// TwinCAT 3 PLC project Lynus_Energy_MRTU
// Title: Lynus Energy ModbusRTU
// Company: Lynus AG
// ProjectVersion: 1.0.0.0
// ProgramVersion: 3.1.4024.12
// libraries:
//   Lynus Persistent Data V1, * (Lynus AG)
//   Lynus Standards, * (EfficientIO)
//   Tc2_Math, * (Beckhoff Automation GmbH)
//   Tc2_ModbusRTU, * (Beckhoff Automation GmbH)
//   Tc2_SerialCom, * (Beckhoff Automation GmbH)
//   Tc2_Standard, * (Beckhoff Automation GmbH)
//   Tc2_System, * (Beckhoff Automation GmbH)
//   Tc3_Module, * (Beckhoff Automation GmbH)
// project tree:
//   DUTs/Delta Inverter/ ST_DeltaPvInverter_Data.TcDUT
//   ENUMs/Delta Inverter/ eDeltaEvent.TcDUT, eDeltaOperatingState.TcDUT
//   ENUMs/Schrack/ E_Schrack_ECS_Error.TcDUT
//   FBs/Delta/ FB_Delta_PV_Inverter_Sunspec.TcPOU
//   FBs/Modbus RTU Master/ FB_KL6xxx_ModbusRTU_22B_Master.TcPOU
//   FBs/Schrack/ FB_ECS_Schrack_EM_CionHome.TcPOU

// ---- DUTs/Delta Inverter/ST_DeltaPvInverter_Data.TcDUT
TYPE ST_DeltaPvInverter_Data :
STRUCT
	eOperatingState			: eDeltaOperatingState;		//Operating State
	eEvent1					: eDeltaEvent;				//Eventfield
	rTotalMPPTPower			: REAL;						//Total DC Power in kW from the MPPT
	rCabinetTemp			: REAL;						//Cabinet Temperature
	rHeatSinkTemp			: REAL;						//Heat Sink Temperature
	arrCurrentFault			: ARRAY[1..8] OF WORD;		//Bit map for the current event of fault on inverter
	arrCurrentError			: ARRAY[1..5] OF WORD;		//Bit map for the current event of error on inverter
	arrCurrentWarning		: ARRAY[1..3] OF WORD;		//Bit map for the current event of warning on inverter
	arrMPPTPower			: ARRAY[1..6] OF REAL;		//Each MPPT DC Power in kW (Max 6 MPPT)
END_STRUCT
END_TYPE

// ---- ENUMs/Delta Inverter/eDeltaEvent.TcDUT
{attribute 'qualified_only'}
{attribute 'strict'}
TYPE eDeltaEvent :
(
	eNoInfo						:= 0,
	eGroundFault				:= 1,
	eDCOverVolt					:= 2,
	eACDisconnect				:= 3,
	eDCDisconnect				:= 4,
	eGridDisconnect				:= 5,
	eCabinetOpen				:= 6,
	eManualShutdown				:= 7,
	eOverTemp					:= 8,
	eOverFrequency				:= 9,
	eUnderFrequency				:= 10,
	eACOverVolt					:= 11,
	eACUnderVolt				:= 12,
	eBlownStringFuse			:= 13,
	eUnderTemp					:= 14,
	eMemoryLoss					:= 15,
	eHWTestFailure				:= 16,
	eOtherAlarm					:= 17,
	eOtherWarning				:= 18
);
END_TYPE

// ---- ENUMs/Delta Inverter/eDeltaOperatingState.TcDUT
{attribute 'qualified_only'}
{attribute 'strict'}
TYPE eDeltaOperatingState :
(
	eNoInfo				:= 0,
	eOff				:= 1,
	eSleeping			:= 2,
	eStarting			:= 3,
	eMppt				:= 4,
	eThrottled			:= 5,
	eShuttingDown		:= 6,
	eFault				:= 7,
	eStandby			:= 8
);
END_TYPE

// ---- ENUMs/Schrack/E_Schrack_ECS_Error.TcDUT
{attribute 'qualified_only'}
{attribute 'strict'}
TYPE E_Schrack_ECS_Error :
(
	eNoError := 0,
	eGroupError := 1,
	eFILSError := 2,
	eChargingCableError := 3,
	eChargingCableRejectedError := 4,
	eLoadContactorError := 5,
	eCommunicationErrorToTheCar := 6,
	eConfigurationErrorOnLP := 7,
	eRCMUError := 8,
	eRCMUErrorCurrentDetected := 9,
	eLockingError := 10,
	eUndervoltageError := 11,
	eOvervoltageError := 12,
	eControllerError := 13
);
END_TYPE

// ---- FBs/Delta/FB_Delta_PV_Inverter_Sunspec.TcPOU
FUNCTION_BLOCK FB_Delta_PV_Inverter_Sunspec
VAR_INPUT PERSISTENT
	bEnable										: BOOL;																			//{#lynus.ag#()} //Enable the Fuctionblock and his logic
	byMBAdress									: BYTE;																			//The Modbus Adress from the Slave
	diNrOfMBRTUMasterLine_IN					: DINT;																			//Number of the RTU Master Function on what this function can send or write data
END_VAR
VAR_OUTPUT
	stDeltaInverterData							: ST_DeltaPvInverter_Data;														//Structure with specific Delta Inverter Data
	stDataEMPower_PV							: ST_ElectricMeter_Output_Power;												//Output structure with Data from Electric Meter PV (Power Data)
	stDataEMCounter_PV							: ST_ElectricMeter_Output_Counter;												//Output structure with Data from Electric Meter PV (Counter Data)
	diNrOfEM_OUT_PV								: DINT;																			//Active Number from the Electric Meter for using on other functions
END_VAR
VAR
	{attribute 'hide'}
	fbElMeter									: FB_ElectricMeter;																//Electric Meter Function 
	{attribute 'hide'}
	fbNumberDevice								: FB_NumberOfDevice;															//Function block to calcualte the number of the Device
	{attribute 'hide'}
	timDelay									: TON;																			//Timer for Delay between Requests
	{attribute 'hide'}
	timTimeout									: TON;																			//Timer for Timeout
	{attribute 'hide'}
	timDissableFunctions						: TON;																			//Timer to dissable the Function after Lynus_Standards.Constants_General.tTimeDissableLynusFunctions Days without connection to the Lynus Cloud
	{attribute 'hide'}
	timResetConnectionOnGVL						: TON;																			//Timer to try reset the connection Flag on the GVL. (When somebody delete the Connection Function and make only a onlinechange)
	{attribute 'hide'}
	FPErrorMaster								: R_TRIG;																		//Internal positive Edge
	{attribute 'hide'}
	FPEnable									: R_TRIG;																		//Internal positive Edge
	{attribute 'hide'}
	fbConvertWord								: FB_CV_WORD_TO_DWORD;															//Convert 2 WORD in a DWORD
	{attribute 'hide'}
	arrPD										: ARRAY[1..5] OF FB_PersistentData_Number;										//Function to save persistent data
	{attribute 'hide'}
	arrDefaultModbusAdress						: ARRAY[1..247] OF BYTE;														//Default Modbuss Adress Array to fill in in the GVL Array after a Online change
	{attribute 'hide'}
	arrDefaultReadWrite							: ARRAY[1..Constants_Bussystems.wQuantityOfRegistersMBRTUMaster] OF WORD;		//Default Read/Write Array to fill in in the GVL Array after a Online change
	{attribute 'hide'}
	arrCounterForGVL							: ARRAY[1..2] OF DINT;															//Counter to clean old data on GVL
	{attribute 'hide'}
	bAdressIsSet								: BOOL;																			//Its true when the new Modbus Adress from the Slave is set in the Array on the GVL for the Master	
	{attribute 'hide'}
	bErrorInverter								: BOOL;																			//Error or Fault from Inverter
	{attribute 'hide'}
	bWarningInverter							: BOOL;																			//Warning from Inverter
	{attribute 'hide'}
	byWaitInStep								: BYTE;																			//Wait in Step before start to clean data on PLC
	{attribute 'hide'}
	byNumberOfSameMBAdress						: BYTE;																			//Number of Same Modbus adress on 1 Modbus Master
	{attribute 'hide'}
	byMBAdress_Old								: BYTE;																			//Old Modbus Adress to compare with the new Modbus Adress to start the state machine to set in the Array on the GVL
	{attribute 'hide'}
	byMBAdress_CP								: BYTE;																			//Variable to compare the Modbus Adress in the State Machine. When the Adress change when the state machine is active then the state machine starts from new with the new adress 
	{attribute 'hide'}
	byLPSlaveAdress								: BYTE;																			//Loop for the state machine to set the adress from the Slave in the array on the GVL
	{attribute 'hide'}
	byLPFillDefaultData							: BYTE;																			//Variable for Loop to fill default values in the Delta output structure
	{attribute 'hide'}
	byLPVendor64062								: BYTE;																			//Variable for Loop to fill the Error,Warning and Faults from Vendor 64062 to the Delta output structure
	{attribute 'hide'}
	iStateGVLData								: INT;																			//State machine to handle the data on the GVL
	{attribute 'hide'}
	iStateModbusRead							: INT;																			//State machine for read out Data over Modbus RTU
	{attribute 'hide'}
	iStateModbusError							: INT;																			//State machine for error out Data over Modbus RTU	
	{attribute 'hide'}
	iStateModbus_CP								: INT;																			//Variable to compare the state machine variable to set or reset the timeout timer
	{attribute 'hide'}
	iSFPowerMPPT								: INT;																			//Scale Factor for MPPT Power
	{attribute 'hide'}
	wNumberOfMPPT								: WORD;																			//Number of MPPT
	{attribute 'hide'}
	wLPCleanBuffer								: WORD;																			//Loop to clear the send and write Buffer on the GVL
	{attribute 'hide'}
	wLPPowerMPPT								: WORD;																			//Variable for Loop to fill the power for each MPPT in the output structure
	{attribute 'hide'}
	wNextModbusStartAdress						: WORD;																			//Next Modbus Start Adress why in Pic 160 the Number of Registers is variabel and so the next Modbus Registers in the next Pics can be different
	{attribute 'hide'}
	wNumberOfInputs								: WORD;																			//Number of Inputs from Pic 401 to calculate the Next Modbus Start Adress
	{attribute 'hide'}
	wPicID										: WORD;																			//ID of the PIC
	{attribute 'hide'}
	diNrOfMBRTUMasterLine_IN_Old				: DINT;																			//Old Modbus RTU Line to compare with the new Modbus RTU Line to start the state machine to set in the Array on the GVL
	{attribute 'hide'}
	diNrOfMBRTUMasterLine_IN_CP					: DINT;																			//Variable to compare the Modbus RTU Line in the State Machine. When the Modbus RTU Line change when the state machine is active then the state machine starts from new with the new Modbus RTU Line
	{attribute 'hide'}
	lrRestNextAdress							: LREAL;																		//Rest of the calculation for new Star Adress. In Sunspec each new PIC start with a even adress
END_VAR
VAR PERSISTENT
	{attribute 'conditionalshow'}
	byMBAdress_ForChange						: BYTE;																			//When we have 2 same Adresses on 1 Modbus RTU Line the byMBAdress_Int is set to 0. After a other change on the Input Adress Field so we can start to set the Adress in the Array in the GVL
	byMBAdress_Int								: BYTE;																			//Internal Adress what is using for the Read and Write functions
END_VAR

//Creator : Kai Ebensperger
//Company : Lynus AG
//Date : 26.10.2021
//Version : 1.0.0.0

//With this function its possible to read out values from the Delta PV Inverter over Modbus RTU
//The Protocoll is the Sunspec Protocol
//Versions that are supported : 1.16
//This Function use the INT+Scalfactor Format

//Infos for Operating State


//NOTE for diNr.....Designation => 
//_IN = Here Data come in from other Functions or go out to other functions about the GVL
//_OUT = Here Data go out to other functions about the GVL

(*--------------------------------------------------------------------------------------------Limits-------------------------------------------------------------------------------------*)

byMBAdress := LIMIT(0,byMBAdress,247);
	diNrOfMBRTUMasterLine_IN := LIMIT(0,diNrOfMBRTUMasterLine_IN,Constants_Bussystems.diMaxNumberOfMBRTUMasterKL6xxx);	

(*-------------------------------------------------------------Calcualte the number of ECS---------------------------------------------------------------*)

fbNumberDevice(
	diActualNumberOfDevices:= Lynus_Standards.GVL_Energy.stNumberOfDevices.diNumberOfElectricMeters, 
	diMaxNumberOfDevices:= Constants_Energy.diMaxNumberOfElectricMeters, 
	udiCounterOnlineChange:= TwinCAT_SystemInfoVarList._AppInfo.OnlineChangeCnt, 
	bNumberIsCalculatet=> , 
	bFPNumberIsCalculatet=> , 
	bOnlineChange=> , 
	diNumberForThisDevice=> diNrOfEM_OUT_PV, 
	diNumberOfTotalDevices=> );

//Write new Numer on GVL
IF fbNumberDevice.bFPNumberIsCalculatet THEN
	Lynus_Standards.GVL_Energy.stNumberOfDevices.diNumberOfElectricMeters := fbNumberDevice.diNumberOfTotalDevices;	
END_IF 

//Delete old Number on GVL
IF fbNumberDevice.bOnlineChange THEN 
	Lynus_Standards.GVL_Energy.stNumberOfDevices.diNumberOfElectricMeters := diNrOfEM_OUT_PV;	
		iStateGVLData := 1;	
			byMBAdress_Old := 0;
				diNrOfMBRTUMasterLine_IN_Old := 0;
END_IF

(*-------------------------------------------------------------Service from Backend is ready and check the connection to backen for dissabel/enable Function---------------------------------------------------------------*)

//Try to reset the variable for connection on the GVL. When all is normal then the Lynus Mqtt connection function set this variable to true in the next cycle
//When we have no connection to the backend then after Lynus_Standards.Constants_General.tTimeDissableLynusFunctions days the Function is dissabled with all of his functionalities
timResetConnectionOnGVL(IN:= NOT timResetConnectionOnGVL.Q, PT:= T#1H, Q=> , ET=> );
	IF timResetConnectionOnGVL.Q THEN Lynus_Standards.GVL_Communicator.bStateConnectionToEnableFunctions := FALSE; END_IF
		IF NOT Lynus_Standards.GVL_Communicator.bStateConnectionToEnableFunctions THEN timDissableFunctions.IN := TRUE; ELSE timDissableFunctions.IN := FALSE; END_IF  
			timDissableFunctions(IN:= , PT:= Lynus_Standards.Constants_General.tTimeDissableLynusFunctions, Q=> , ET=> );
			
(*--------------------------------------------------------------------------------------------Error from the Master Function-------------------------------------------------------------------------------------*)

FPErrorMaster(CLK:= Lynus_Standards.GVL_Bussystems.stDataOfMBRTUMasterKL6xxx[diNrOfMBRTUMasterLine_IN].byErrorWarning = 2 AND bEnable, Q=> );

(*--------------------------------------------------------------------------------------------Modbus Adress Slave Function-------------------------------------------------------------------------------------*)

FPEnable(CLK:= bEnable, Q=> );

//When the Adress is changed then set the new Adress in the Array
//When we have the Adress more then 1 time in 1 line then set to 0 and wait for the next change on the Input Variable for the Modbus Adress
IF byMBAdress <> byMBAdress_ForChange AND bEnable THEN byMBAdress_ForChange := byMBAdress; byNumberOfSameMBAdress := 0; END_IF     
	IF byMBAdress <> byMBAdress_Int AND byNumberOfSameMBAdress = 0 AND bEnable THEN byMBAdress_Int := byMBAdress; END_IF 
		IF NOT bEnable THEN byMBAdress_Int := 0; END_IF 
		
IF NOT Lynus_Standards.GVL_Bussystems.stDataOfMBRTUMasterKL6xxx[diNrOfMBRTUMasterLine_IN].bNoNewMBusAdress AND iStateGVLData = 0 AND (MEMCMP(ADR(byMBAdress_Int),ADR(byMBAdress_Old),SIZEOF(byMBAdress_Old)) <> 0 OR MEMCMP(ADR(diNrOfMBRTUMasterLine_IN),ADR(diNrOfMBRTUMasterLine_IN_Old),SIZEOF(diNrOfMBRTUMasterLine_IN_Old)) <> 0) THEN
	//Check if we have more then 1 time this Adress in 1 Line
	byNumberOfSameMBAdress := 0;	
		FOR byLPSlaveAdress := 1 TO 247 BY 1 DO
			IF Lynus_Standards.GVL_Bussystems.stDataOfMBRTUMasterKL6xxx[diNrOfMBRTUMasterLine_IN].arrAllModbusSlaveAdresses[byLPSlaveAdress] = byMBAdress_Int AND 
					Lynus_Standards.GVL_Bussystems.stDataOfMBRTUMasterKL6xxx[diNrOfMBRTUMasterLine_IN].arrAllModbusSlaveAdresses[byLPSlaveAdress] <> 0 THEN 
						byNumberOfSameMBAdress := byNumberOfSameMBAdress + 1; 
				END_IF 
		END_FOR
			IF byNumberOfSameMBAdress > 0 THEN 
				byMBAdress_Int := 0;
			END_IF	
				bAdressIsSet := FALSE; 
					//Delte the old Adress from the old Array
					FOR byLPSlaveAdress := 1 TO 247 BY 1 DO
						IF Lynus_Standards.GVL_Bussystems.stDataOfMBRTUMasterKL6xxx[diNrOfMBRTUMasterLine_IN_Old].arrAllModbusSlaveAdresses[byLPSlaveAdress] = byMBAdress_Old THEN
							Lynus_Standards.GVL_Bussystems.stDataOfMBRTUMasterKL6xxx[diNrOfMBRTUMasterLine_IN_Old].arrAllModbusSlaveAdresses[byLPSlaveAdress] := 0;
						END_IF	 
					END_FOR
						//Set the New Adress in Array
						byMBAdress_Old := byMBAdress_Int;
							diNrOfMBRTUMasterLine_IN_Old := diNrOfMBRTUMasterLine_IN;
								FOR byLPSlaveAdress := 1 TO 247 BY 1 DO
									IF Lynus_Standards.GVL_Bussystems.stDataOfMBRTUMasterKL6xxx[diNrOfMBRTUMasterLine_IN].arrAllModbusSlaveAdresses[byLPSlaveAdress] = 0 AND NOT bAdressIsSet THEN 
										Lynus_Standards.GVL_Bussystems.stDataOfMBRTUMasterKL6xxx[diNrOfMBRTUMasterLine_IN].arrAllModbusSlaveAdresses[byLPSlaveAdress] := byMBAdress_Int; 
											bAdressIsSet := TRUE;
									END_IF 
								END_FOR
END_IF	

(*--------------------------------------------------------------------------------------------State Machine Read--------------------------------------------------------------------------------------*)

//Timer for Delay
timDelay(IN:= , PT:= T#250MS, Q=> , ET=> );

//Timer for Timeout in Statemachine
IF iStateModbusRead > 0 AND iStateModbusRead <= 8 AND iStateModbusRead = iStateModbus_CP THEN
		timTimeout.IN := TRUE;
ELSE	
		timTimeout.IN := FALSE;
END_IF
	//Timeout Timer is dissabled when the slave wait that his adress is in porgress on the RTU Master, or is dissabled or the Terminal is not configured
	IF iStateModbusRead = 0 OR NOT bEnable OR NOT Lynus_Standards.GVL_Bussystems.stDataOfMBRTUMasterKL6xxx[diNrOfMBRTUMasterLine_IN].bTerminalIsConfigured THEN timTimeout.IN := FALSE; END_IF
		timTimeout(IN:= , PT:= T#15S, Q=> , ET=> );

//Not Enabled
IF NOT bEnable OR NOT Lynus_Standards.GVL_Bussystems.stDataOfMBRTUMasterKL6xxx[diNrOfMBRTUMasterLine_IN].bTerminalIsConfigured THEN iStateModbusRead := 0; iStateModbusError := 0; END_IF		
		
CASE iStateModbusRead OF

	0://Init Step (Wait that the Slave is enabled and the Terminal is configured)
		
		//Set Delta Output Structure to default
		IF NOT bEnable OR NOT Lynus_Standards.GVL_Bussystems.stDataOfMBRTUMasterKL6xxx[diNrOfMBRTUMasterLine_IN].bTerminalIsConfigured THEN 
			stDeltaInverterData.rTotalMPPTPower := 0;
				stDeltaInverterData.rCabinetTemp := 0;
					stDeltaInverterData.rHeatSinkTemp := 0;
						FOR byLPFillDefaultData := 1 TO 6 BY 1 DO
							stDeltaInverterData.arrMPPTPower[byLPFillDefaultData] := 0;
						END_FOR
							stDeltaInverterData.eEvent1 := eDeltaEvent.eNoInfo;
								stDeltaInverterData.eOperatingState := eDeltaOperatingState.eNoInfo;
		END_IF
		
		iSFPowerMPPT := 0;
			wNumberOfMPPT := 0;
				wNextModbusStartAdress := 0;
					wNumberOfInputs := 0;
						lrRestNextAdress := 0;
				
		IF bEnable AND Lynus_Standards.GVL_Bussystems.stDataOfMBRTUMasterKL6xxx[diNrOfMBRTUMasterLine_IN].bTerminalIsConfigured THEN
			//Start Timer for start the Statemachine
			IF NOT Lynus_Standards.GVL_Bussystems.stDataOfMBRTUMasterKL6xxx[diNrOfMBRTUMasterLine_IN].bMasterIsBusy THEN timDelay.IN := TRUE; END_IF 
		
			//Reset the Read and Write Buffer on the GVL before starting
			IF byMBAdress_Int = Lynus_Standards.GVL_Bussystems.stDataOfMBRTUMasterKL6xxx[diNrOfMBRTUMasterLine_IN].byActualMBAdressInProgrss THEN
				FOR wLPCleanBuffer := 1 TO Constants_Bussystems.wQuantityOfRegistersMBRTUMaster BY 1 DO
					Lynus_Standards.GVL_Bussystems.stDataOfMBRTUMasterKL6xxx[diNrOfMBRTUMasterLine_IN].arrReadOutData[wLPCleanBuffer] := 0;
						Lynus_Standards.GVL_Bussystems.stDataOfMBRTUMasterKL6xxx[diNrOfMBRTUMasterLine_IN].arrWriteOutData[wLPCleanBuffer] := 0;
				END_FOR
			END_IF
			
			IF timDelay.Q AND byMBAdress_Int = Lynus_Standards.GVL_Bussystems.stDataOfMBRTUMasterKL6xxx[diNrOfMBRTUMasterLine_IN].byActualMBAdressInProgrss AND NOT Lynus_Standards.GVL_Bussystems.stDataOfMBRTUMasterKL6xxx[diNrOfMBRTUMasterLine_IN].bReadWriteIsDone THEN
				timDelay.IN := FALSE;
					iStateModbusRead := 1;
						diNrOfMBRTUMasterLine_IN_CP := diNrOfMBRTUMasterLine_IN;
							byMBAdress_CP := byMBAdress_Int; 	
								Lynus_Standards.GVL_Bussystems.stDataOfMBRTUMasterKL6xxx[diNrOfMBRTUMasterLine_IN].bSlaveStartReadOrWrite := FALSE;
			END_IF
		END_IF
	
	1://Read Out Values from Pic 103 of the Sunspec Protocol (Register 40084)
		iStateModbus_CP := iStateModbusRead;
		
		Lynus_Standards.GVL_Bussystems.stDataOfMBRTUMasterKL6xxx[diNrOfMBRTUMasterLine_IN].eMBRTUReadWriteMode := E_MBRTUMaster_ReadWriteMode.eModbusRTUMaster_ReadRegs;
			Lynus_Standards.GVL_Bussystems.stDataOfMBRTUMasterKL6xxx[diNrOfMBRTUMasterLine_IN].wNumberOfRegister := 39;
				Lynus_Standards.GVL_Bussystems.stDataOfMBRTUMasterKL6xxx[diNrOfMBRTUMasterLine_IN].wModbusRegister := 40073;
		
		IF NOT Lynus_Standards.GVL_Bussystems.stDataOfMBRTUMasterKL6xxx[diNrOfMBRTUMasterLine_IN].bMasterIsBusy THEN timDelay.IN := TRUE; END_IF 

		//Copy the read out Data
		IF NOT Lynus_Standards.GVL_Bussystems.stDataOfMBRTUMasterKL6xxx[diNrOfMBRTUMasterLine_IN].bMasterIsBusy AND Lynus_Standards.GVL_Bussystems.stDataOfMBRTUMasterKL6xxx[diNrOfMBRTUMasterLine_IN].byErrorWarning = 0 AND timDelay.Q AND diNrOfMBRTUMasterLine_IN = diNrOfMBRTUMasterLine_IN_CP AND byMBAdress_Int = byMBAdress_CP THEN
			//Current L1
			IF WORD_TO_INT(Lynus_Standards.GVL_Bussystems.stDataOfMBRTUMasterKL6xxx[diNrOfMBRTUMasterLine_IN].arrReadOutData[4]) >= - 10 AND WORD_TO_INT(Lynus_Standards.GVL_Bussystems.stDataOfMBRTUMasterKL6xxx[diNrOfMBRTUMasterLine_IN].arrReadOutData[4]) <= 10 THEN
				fbElMeter.lrCurrentL1 := Lynus_Standards.GVL_Bussystems.stDataOfMBRTUMasterKL6xxx[diNrOfMBRTUMasterLine_IN].arrReadOutData[1] * EXPT(10,WORD_TO_INT(Lynus_Standards.GVL_Bussystems.stDataOfMBRTUMasterKL6xxx[diNrOfMBRTUMasterLine_IN].arrReadOutData[4]));
			END_IF
			//Current L2
			IF WORD_TO_INT(Lynus_Standards.GVL_Bussystems.stDataOfMBRTUMasterKL6xxx[diNrOfMBRTUMasterLine_IN].arrReadOutData[4]) >= - 10 AND WORD_TO_INT(Lynus_Standards.GVL_Bussystems.stDataOfMBRTUMasterKL6xxx[diNrOfMBRTUMasterLine_IN].arrReadOutData[4]) <= 10 THEN
				fbElMeter.lrCurrentL2 := Lynus_Standards.GVL_Bussystems.stDataOfMBRTUMasterKL6xxx[diNrOfMBRTUMasterLine_IN].arrReadOutData[2] * EXPT(10,WORD_TO_INT(Lynus_Standards.GVL_Bussystems.stDataOfMBRTUMasterKL6xxx[diNrOfMBRTUMasterLine_IN].arrReadOutData[4]));
			END_IF
			//Current L3
			IF WORD_TO_INT(Lynus_Standards.GVL_Bussystems.stDataOfMBRTUMasterKL6xxx[diNrOfMBRTUMasterLine_IN].arrReadOutData[4]) >= - 10 AND WORD_TO_INT(Lynus_Standards.GVL_Bussystems.stDataOfMBRTUMasterKL6xxx[diNrOfMBRTUMasterLine_IN].arrReadOutData[4]) <= 10 THEN
				fbElMeter.lrCurrentL3 := Lynus_Standards.GVL_Bussystems.stDataOfMBRTUMasterKL6xxx[diNrOfMBRTUMasterLine_IN].arrReadOutData[3] * EXPT(10,WORD_TO_INT(Lynus_Standards.GVL_Bussystems.stDataOfMBRTUMasterKL6xxx[diNrOfMBRTUMasterLine_IN].arrReadOutData[4]));
			END_IF
			//Voltage L1/N
			IF WORD_TO_INT(Lynus_Standards.GVL_Bussystems.stDataOfMBRTUMasterKL6xxx[diNrOfMBRTUMasterLine_IN].arrReadOutData[11]) >= - 10 AND WORD_TO_INT(Lynus_Standards.GVL_Bussystems.stDataOfMBRTUMasterKL6xxx[diNrOfMBRTUMasterLine_IN].arrReadOutData[11]) <= 10 THEN
				fbElMeter.lrVoltageL1N := Lynus_Standards.GVL_Bussystems.stDataOfMBRTUMasterKL6xxx[diNrOfMBRTUMasterLine_IN].arrReadOutData[8] * EXPT(10,WORD_TO_INT(Lynus_Standards.GVL_Bussystems.stDataOfMBRTUMasterKL6xxx[diNrOfMBRTUMasterLine_IN].arrReadOutData[11]));
			END_IF
			//Voltage L2/N
			IF WORD_TO_INT(Lynus_Standards.GVL_Bussystems.stDataOfMBRTUMasterKL6xxx[diNrOfMBRTUMasterLine_IN].arrReadOutData[11]) >= - 10 AND WORD_TO_INT(Lynus_Standards.GVL_Bussystems.stDataOfMBRTUMasterKL6xxx[diNrOfMBRTUMasterLine_IN].arrReadOutData[11]) <= 10 THEN
				fbElMeter.lrVoltageL2N := Lynus_Standards.GVL_Bussystems.stDataOfMBRTUMasterKL6xxx[diNrOfMBRTUMasterLine_IN].arrReadOutData[9] * EXPT(10,WORD_TO_INT(Lynus_Standards.GVL_Bussystems.stDataOfMBRTUMasterKL6xxx[diNrOfMBRTUMasterLine_IN].arrReadOutData[11]));
			END_IF
			//Voltage L3/N
			IF WORD_TO_INT(Lynus_Standards.GVL_Bussystems.stDataOfMBRTUMasterKL6xxx[diNrOfMBRTUMasterLine_IN].arrReadOutData[11]) >= - 10 AND WORD_TO_INT(Lynus_Standards.GVL_Bussystems.stDataOfMBRTUMasterKL6xxx[diNrOfMBRTUMasterLine_IN].arrReadOutData[11]) <= 10 THEN
				fbElMeter.lrVoltageL3N := Lynus_Standards.GVL_Bussystems.stDataOfMBRTUMasterKL6xxx[diNrOfMBRTUMasterLine_IN].arrReadOutData[10] * EXPT(10,WORD_TO_INT(Lynus_Standards.GVL_Bussystems.stDataOfMBRTUMasterKL6xxx[diNrOfMBRTUMasterLine_IN].arrReadOutData[11]));
			END_IF
			//AC Power
			IF WORD_TO_INT(Lynus_Standards.GVL_Bussystems.stDataOfMBRTUMasterKL6xxx[diNrOfMBRTUMasterLine_IN].arrReadOutData[13]) >= - 10 AND WORD_TO_INT(Lynus_Standards.GVL_Bussystems.stDataOfMBRTUMasterKL6xxx[diNrOfMBRTUMasterLine_IN].arrReadOutData[13]) <= 10 THEN  
				fbElMeter.lrPowerTotal := WORD_TO_INT(Lynus_Standards.GVL_Bussystems.stDataOfMBRTUMasterKL6xxx[diNrOfMBRTUMasterLine_IN].arrReadOutData[12]) * EXPT(10,WORD_TO_INT(Lynus_Standards.GVL_Bussystems.stDataOfMBRTUMasterKL6xxx[diNrOfMBRTUMasterLine_IN].arrReadOutData[13]));
			END_IF
			//Hz
			IF WORD_TO_INT(Lynus_Standards.GVL_Bussystems.stDataOfMBRTUMasterKL6xxx[diNrOfMBRTUMasterLine_IN].arrReadOutData[15]) >= - 10 AND WORD_TO_INT(Lynus_Standards.GVL_Bussystems.stDataOfMBRTUMasterKL6xxx[diNrOfMBRTUMasterLine_IN].arrReadOutData[15]) <= 10 THEN  
				fbElMeter.lrFrequency := Lynus_Standards.GVL_Bussystems.stDataOfMBRTUMasterKL6xxx[diNrOfMBRTUMasterLine_IN].arrReadOutData[14] * EXPT(10,WORD_TO_INT(Lynus_Standards.GVL_Bussystems.stDataOfMBRTUMasterKL6xxx[diNrOfMBRTUMasterLine_IN].arrReadOutData[15]));
			END_IF
			//Apparent Power
			IF WORD_TO_INT(Lynus_Standards.GVL_Bussystems.stDataOfMBRTUMasterKL6xxx[diNrOfMBRTUMasterLine_IN].arrReadOutData[17]) >= - 10 AND WORD_TO_INT(Lynus_Standards.GVL_Bussystems.stDataOfMBRTUMasterKL6xxx[diNrOfMBRTUMasterLine_IN].arrReadOutData[17]) <= 10 THEN  
				fbElMeter.lrApparentPowerTotal := WORD_TO_INT(Lynus_Standards.GVL_Bussystems.stDataOfMBRTUMasterKL6xxx[diNrOfMBRTUMasterLine_IN].arrReadOutData[16]) * EXPT(10,WORD_TO_INT(Lynus_Standards.GVL_Bussystems.stDataOfMBRTUMasterKL6xxx[diNrOfMBRTUMasterLine_IN].arrReadOutData[17]));
			END_IF
			//Reactive Power
			IF WORD_TO_INT(Lynus_Standards.GVL_Bussystems.stDataOfMBRTUMasterKL6xxx[diNrOfMBRTUMasterLine_IN].arrReadOutData[19]) >= - 10 AND WORD_TO_INT(Lynus_Standards.GVL_Bussystems.stDataOfMBRTUMasterKL6xxx[diNrOfMBRTUMasterLine_IN].arrReadOutData[19]) <= 10 THEN  
				fbElMeter.lrReactivePowerTotal := WORD_TO_INT(Lynus_Standards.GVL_Bussystems.stDataOfMBRTUMasterKL6xxx[diNrOfMBRTUMasterLine_IN].arrReadOutData[18]) * EXPT(10,WORD_TO_INT(Lynus_Standards.GVL_Bussystems.stDataOfMBRTUMasterKL6xxx[diNrOfMBRTUMasterLine_IN].arrReadOutData[19]));
			END_IF
			//Produced Energy
			IF WORD_TO_INT(Lynus_Standards.GVL_Bussystems.stDataOfMBRTUMasterKL6xxx[diNrOfMBRTUMasterLine_IN].arrReadOutData[24]) >= - 10 AND WORD_TO_INT(Lynus_Standards.GVL_Bussystems.stDataOfMBRTUMasterKL6xxx[diNrOfMBRTUMasterLine_IN].arrReadOutData[24]) <= 10 THEN  
				fbConvertWord(wInputValue_1:= Lynus_Standards.GVL_Bussystems.stDataOfMBRTUMasterKL6xxx[diNrOfMBRTUMasterLine_IN].arrReadOutData[22], wInputValue_2:= Lynus_Standards.GVL_Bussystems.stDataOfMBRTUMasterKL6xxx[diNrOfMBRTUMasterLine_IN].arrReadOutData[23], eByteOrderForConvert:= eByteOrder.eBigEndian, dwOutputValue=> );
					fbElMeter.lrCounterEnergyT1_Production := fbConvertWord.dwOutputValue * EXPT(10,WORD_TO_INT(Lynus_Standards.GVL_Bussystems.stDataOfMBRTUMasterKL6xxx[diNrOfMBRTUMasterLine_IN].arrReadOutData[24]));
						fbElMeter.lrCounterEnergyT1_Production := fbElMeter.lrCounterEnergyT1_Production / 1000;
							fbElMeter.lrTotalCounterEnergy_Production := fbElMeter.lrCounterEnergyT1_Production; 	
			END_IF
			//Cabinet Temperature
			IF WORD_TO_INT(Lynus_Standards.GVL_Bussystems.stDataOfMBRTUMasterKL6xxx[diNrOfMBRTUMasterLine_IN].arrReadOutData[35]) >= - 10 AND WORD_TO_INT(Lynus_Standards.GVL_Bussystems.stDataOfMBRTUMasterKL6xxx[diNrOfMBRTUMasterLine_IN].arrReadOutData[35]) <= 10 THEN  
				stDeltaInverterData.rCabinetTemp := LREAL_TO_REAL(WORD_TO_INT(Lynus_Standards.GVL_Bussystems.stDataOfMBRTUMasterKL6xxx[diNrOfMBRTUMasterLine_IN].arrReadOutData[31]) * EXPT(10,WORD_TO_INT(Lynus_Standards.GVL_Bussystems.stDataOfMBRTUMasterKL6xxx[diNrOfMBRTUMasterLine_IN].arrReadOutData[35])));
			END_IF
			//Heat Sink Temperature
			IF WORD_TO_INT(Lynus_Standards.GVL_Bussystems.stDataOfMBRTUMasterKL6xxx[diNrOfMBRTUMasterLine_IN].arrReadOutData[35]) >= - 10 AND WORD_TO_INT(Lynus_Standards.GVL_Bussystems.stDataOfMBRTUMasterKL6xxx[diNrOfMBRTUMasterLine_IN].arrReadOutData[35]) <= 10 THEN  
				stDeltaInverterData.rHeatSinkTemp := LREAL_TO_REAL(WORD_TO_INT(Lynus_Standards.GVL_Bussystems.stDataOfMBRTUMasterKL6xxx[diNrOfMBRTUMasterLine_IN].arrReadOutData[32]) * EXPT(10,WORD_TO_INT(Lynus_Standards.GVL_Bussystems.stDataOfMBRTUMasterKL6xxx[diNrOfMBRTUMasterLine_IN].arrReadOutData[35])));
			END_IF
			//Operating State
			stDeltaInverterData.eOperatingState := eDeltaOperatingState.eNoInfo;
			IF Lynus_Standards.GVL_Bussystems.stDataOfMBRTUMasterKL6xxx[diNrOfMBRTUMasterLine_IN].arrReadOutData[36] = 1 THEN stDeltaInverterData.eOperatingState := eDeltaOperatingState.eOff;
			ELSIF Lynus_Standards.GVL_Bussystems.stDataOfMBRTUMasterKL6xxx[diNrOfMBRTUMasterLine_IN].arrReadOutData[36] = 2 THEN stDeltaInverterData.eOperatingState := eDeltaOperatingState.eSleeping;
			ELSIF Lynus_Standards.GVL_Bussystems.stDataOfMBRTUMasterKL6xxx[diNrOfMBRTUMasterLine_IN].arrReadOutData[36] = 3 THEN stDeltaInverterData.eOperatingState := eDeltaOperatingState.eStarting;
			ELSIF Lynus_Standards.GVL_Bussystems.stDataOfMBRTUMasterKL6xxx[diNrOfMBRTUMasterLine_IN].arrReadOutData[36] = 4 THEN stDeltaInverterData.eOperatingState := eDeltaOperatingState.eMppt;
			ELSIF Lynus_Standards.GVL_Bussystems.stDataOfMBRTUMasterKL6xxx[diNrOfMBRTUMasterLine_IN].arrReadOutData[36] = 5 THEN stDeltaInverterData.eOperatingState := eDeltaOperatingState.eThrottled;
			ELSIF Lynus_Standards.GVL_Bussystems.stDataOfMBRTUMasterKL6xxx[diNrOfMBRTUMasterLine_IN].arrReadOutData[36] = 6 THEN stDeltaInverterData.eOperatingState := eDeltaOperatingState.eShuttingDown;
			ELSIF Lynus_Standards.GVL_Bussystems.stDataOfMBRTUMasterKL6xxx[diNrOfMBRTUMasterLine_IN].arrReadOutData[36] = 7 THEN stDeltaInverterData.eOperatingState := eDeltaOperatingState.eFault;
			ELSIF Lynus_Standards.GVL_Bussystems.stDataOfMBRTUMasterKL6xxx[diNrOfMBRTUMasterLine_IN].arrReadOutData[36] = 8 THEN stDeltaInverterData.eOperatingState := eDeltaOperatingState.eStandby;
			END_IF 
			//Event 1
			fbConvertWord(wInputValue_1:= Lynus_Standards.GVL_Bussystems.stDataOfMBRTUMasterKL6xxx[diNrOfMBRTUMasterLine_IN].arrReadOutData[38], wInputValue_2:= Lynus_Standards.GVL_Bussystems.stDataOfMBRTUMasterKL6xxx[diNrOfMBRTUMasterLine_IN].arrReadOutData[39], eByteOrderForConvert:= eByteOrder.eBigEndian, dwOutputValue=> );
			stDeltaInverterData.eEvent1 := eDeltaEvent.eNoInfo;
			IF fbConvertWord.dwOutputValue.0 THEN stDeltaInverterData.eEvent1 := eDeltaEvent.eGroundFault;
			ELSIF fbConvertWord.dwOutputValue.1 THEN stDeltaInverterData.eEvent1 := eDeltaEvent.eDCOverVolt;
			ELSIF fbConvertWord.dwOutputValue.2 THEN stDeltaInverterData.eEvent1 := eDeltaEvent.eACDisconnect;
			ELSIF fbConvertWord.dwOutputValue.3 THEN stDeltaInverterData.eEvent1 := eDeltaEvent.eDCDisconnect;
			ELSIF fbConvertWord.dwOutputValue.4 THEN stDeltaInverterData.eEvent1 := eDeltaEvent.eGridDisconnect;
			ELSIF fbConvertWord.dwOutputValue.5 THEN stDeltaInverterData.eEvent1 := eDeltaEvent.eCabinetOpen;
			ELSIF fbConvertWord.dwOutputValue.6 THEN stDeltaInverterData.eEvent1 := eDeltaEvent.eManualShutdown;
			ELSIF fbConvertWord.dwOutputValue.7 THEN stDeltaInverterData.eEvent1 := eDeltaEvent.eOverTemp;
			ELSIF fbConvertWord.dwOutputValue.8 THEN stDeltaInverterData.eEvent1 := eDeltaEvent.eOverFrequency;
			ELSIF fbConvertWord.dwOutputValue.9 THEN stDeltaInverterData.eEvent1 := eDeltaEvent.eUnderFrequency;
			ELSIF fbConvertWord.dwOutputValue.10 THEN stDeltaInverterData.eEvent1 := eDeltaEvent.eACOverVolt;
			ELSIF fbConvertWord.dwOutputValue.11 THEN stDeltaInverterData.eEvent1 := eDeltaEvent.eACUnderVolt;
			ELSIF fbConvertWord.dwOutputValue.12 THEN stDeltaInverterData.eEvent1 := eDeltaEvent.eBlownStringFuse;
			ELSIF fbConvertWord.dwOutputValue.13 THEN stDeltaInverterData.eEvent1 := eDeltaEvent.eUnderTemp;
			ELSIF fbConvertWord.dwOutputValue.14 THEN stDeltaInverterData.eEvent1 := eDeltaEvent.eMemoryLoss;
			ELSIF fbConvertWord.dwOutputValue.15 THEN stDeltaInverterData.eEvent1 := eDeltaEvent.eHWTestFailure;
			ELSIF fbConvertWord.dwOutputValue.16 THEN stDeltaInverterData.eEvent1 := eDeltaEvent.eOtherAlarm;
			ELSIF fbConvertWord.dwOutputValue.17 THEN stDeltaInverterData.eEvent1 := eDeltaEvent.eOtherWarning;	
			END_IF
		END_IF     				
		
		//Send the Read or Write Command to the Master
		Lynus_Standards.GVL_Bussystems.stDataOfMBRTUMasterKL6xxx[diNrOfMBRTUMasterLine_IN].bSlaveStartReadOrWrite := TRUE;
		
		//Go to the Next Step
		IF NOT Lynus_Standards.GVL_Bussystems.stDataOfMBRTUMasterKL6xxx[diNrOfMBRTUMasterLine_IN].bMasterIsBusy AND Lynus_Standards.GVL_Bussystems.stDataOfMBRTUMasterKL6xxx[diNrOfMBRTUMasterLine_IN].byErrorWarning = 0 AND timDelay.Q AND 
			diNrOfMBRTUMasterLine_IN = diNrOfMBRTUMasterLine_IN_CP AND byMBAdress_Int = byMBAdress_CP AND NOT timTimeout.Q THEN
				timDelay.IN := FALSE;
					Lynus_Standards.GVL_Bussystems.stDataOfMBRTUMasterKL6xxx[diNrOfMBRTUMasterLine_IN].bSlaveStartReadOrWrite := FALSE;
						iStateModbusRead := 2;
							wNextModbusStartAdress := 40122;		
		END_IF

			//Error on Master, changes on Inputs or Timeout
		 	IF timTimeout.Q OR diNrOfMBRTUMasterLine_IN <> diNrOfMBRTUMasterLine_IN_CP OR byMBAdress_Int <> byMBAdress_CP OR FPErrorMaster.Q THEN 
				iStateModbusError := 300; 
					diNrOfMBRTUMasterLine_IN_CP := diNrOfMBRTUMasterLine_IN; 
						byMBAdress_CP := byMBAdress_Int; 
			END_IF 
	
	2://Read Out Values from Pic 120 to Start Adress for PIC 160 of the Sunspec Protocoll		
		iStateModbus_CP := iStateModbusRead;
		
		Lynus_Standards.GVL_Bussystems.stDataOfMBRTUMasterKL6xxx[diNrOfMBRTUMasterLine_IN].eMBRTUReadWriteMode := E_MBRTUMaster_ReadWriteMode.eModbusRTUMaster_ReadRegs;
			Lynus_Standards.GVL_Bussystems.stDataOfMBRTUMasterKL6xxx[diNrOfMBRTUMasterLine_IN].wNumberOfRegister := 2;
				Lynus_Standards.GVL_Bussystems.stDataOfMBRTUMasterKL6xxx[diNrOfMBRTUMasterLine_IN].wModbusRegister := wNextModbusStartAdress;
		
		IF NOT Lynus_Standards.GVL_Bussystems.stDataOfMBRTUMasterKL6xxx[diNrOfMBRTUMasterLine_IN].bMasterIsBusy THEN timDelay.IN := TRUE; END_IF 

		//Copy the read out Data
		IF NOT Lynus_Standards.GVL_Bussystems.stDataOfMBRTUMasterKL6xxx[diNrOfMBRTUMasterLine_IN].bMasterIsBusy AND Lynus_Standards.GVL_Bussystems.stDataOfMBRTUMasterKL6xxx[diNrOfMBRTUMasterLine_IN].byErrorWarning = 0 AND timDelay.Q AND diNrOfMBRTUMasterLine_IN = diNrOfMBRTUMasterLine_IN_CP AND byMBAdress_Int = byMBAdress_CP THEN
			//PIC ID
			wPicID := Lynus_Standards.GVL_Bussystems.stDataOfMBRTUMasterKL6xxx[diNrOfMBRTUMasterLine_IN].arrReadOutData[1];
			//Number of Inputs
			wNumberOfInputs := Lynus_Standards.GVL_Bussystems.stDataOfMBRTUMasterKL6xxx[diNrOfMBRTUMasterLine_IN].arrReadOutData[2];
		END_IF     					
		
		//Send the Read or Write Command to the Master
		Lynus_Standards.GVL_Bussystems.stDataOfMBRTUMasterKL6xxx[diNrOfMBRTUMasterLine_IN].bSlaveStartReadOrWrite := TRUE;
		
		//Go to the Next Step
		IF NOT Lynus_Standards.GVL_Bussystems.stDataOfMBRTUMasterKL6xxx[diNrOfMBRTUMasterLine_IN].bMasterIsBusy AND Lynus_Standards.GVL_Bussystems.stDataOfMBRTUMasterKL6xxx[diNrOfMBRTUMasterLine_IN].byErrorWarning = 0 AND timDelay.Q AND 
			diNrOfMBRTUMasterLine_IN = diNrOfMBRTUMasterLine_IN_CP AND byMBAdress_Int = byMBAdress_CP AND NOT timTimeout.Q THEN
				timDelay.IN := FALSE;
					Lynus_Standards.GVL_Bussystems.stDataOfMBRTUMasterKL6xxx[diNrOfMBRTUMasterLine_IN].bSlaveStartReadOrWrite := FALSE;
						iStateModbusRead := 3;	
							lrRestNextAdress := 0;
			//Calculate next Modbus Start Adress for next Pic
			wNextModbusStartAdress := wNextModbusStartAdress + wNumberOfInputs + 2;
				lrRestNextAdress := FRAC(WORD_TO_REAL(wNextModbusStartAdress) / 2);	
					//If it ends with an odd number, the next PIC starts with an even address
					IF lrRestNextAdress <> 0 THEN wNextModbusStartAdress := wNextModbusStartAdress + 1; END_IF 
		END_IF

			//Error on Master, changes on Inputs or Timeout
		 	IF timTimeout.Q OR diNrOfMBRTUMasterLine_IN <> diNrOfMBRTUMasterLine_IN_CP OR byMBAdress_Int <> byMBAdress_CP OR FPErrorMaster.Q THEN 
				iStateModbusError := 300; 
					diNrOfMBRTUMasterLine_IN_CP := diNrOfMBRTUMasterLine_IN; 
						byMBAdress_CP := byMBAdress_Int; 
			END_IF		
	
	3://Check the PIC ID
		iStateModbus_CP := iStateModbusRead;
		
		IF wPicID < 160 THEN
			//Back to Step 2
			iStateModbusRead := 2;
		ELSE
			//next Step with values
			iStateModbusRead := 4;
				//Calculate next Modbus Start Adress for next Pic
				wNextModbusStartAdress := wNextModbusStartAdress - wNumberOfInputs - 2;
		END_IF
		
	
	4://Read Out Values from Pic 160 of the Sunspec Protocol
		iStateModbus_CP := iStateModbusRead;
		
		Lynus_Standards.GVL_Bussystems.stDataOfMBRTUMasterKL6xxx[diNrOfMBRTUMasterLine_IN].eMBRTUReadWriteMode := E_MBRTUMaster_ReadWriteMode.eModbusRTUMaster_ReadRegs;
			Lynus_Standards.GVL_Bussystems.stDataOfMBRTUMasterKL6xxx[diNrOfMBRTUMasterLine_IN].wNumberOfRegister := 9;
				Lynus_Standards.GVL_Bussystems.stDataOfMBRTUMasterKL6xxx[diNrOfMBRTUMasterLine_IN].wModbusRegister := wNextModbusStartAdress;
		
		IF NOT Lynus_Standards.GVL_Bussystems.stDataOfMBRTUMasterKL6xxx[diNrOfMBRTUMasterLine_IN].bMasterIsBusy THEN timDelay.IN := TRUE; END_IF 

		//Copy the read out Data
		IF NOT Lynus_Standards.GVL_Bussystems.stDataOfMBRTUMasterKL6xxx[diNrOfMBRTUMasterLine_IN].bMasterIsBusy AND Lynus_Standards.GVL_Bussystems.stDataOfMBRTUMasterKL6xxx[diNrOfMBRTUMasterLine_IN].byErrorWarning = 0 AND timDelay.Q AND diNrOfMBRTUMasterLine_IN = diNrOfMBRTUMasterLine_IN_CP AND byMBAdress_Int = byMBAdress_CP THEN
			//PIC ID
			wPicID := Lynus_Standards.GVL_Bussystems.stDataOfMBRTUMasterKL6xxx[diNrOfMBRTUMasterLine_IN].arrReadOutData[1];
			//Number of Inputs
			wNumberOfInputs := Lynus_Standards.GVL_Bussystems.stDataOfMBRTUMasterKL6xxx[diNrOfMBRTUMasterLine_IN].arrReadOutData[2];
			//Scale Factor for String Power
			iSFPowerMPPT := WORD_TO_INT(Lynus_Standards.GVL_Bussystems.stDataOfMBRTUMasterKL6xxx[diNrOfMBRTUMasterLine_IN].arrReadOutData[5]);
			//Number of MPPT Moduls
			wNumberOfMPPT := Lynus_Standards.GVL_Bussystems.stDataOfMBRTUMasterKL6xxx[diNrOfMBRTUMasterLine_IN].arrReadOutData[9];
		END_IF     				
		
		//Send the Read or Write Command to the Master
		Lynus_Standards.GVL_Bussystems.stDataOfMBRTUMasterKL6xxx[diNrOfMBRTUMasterLine_IN].bSlaveStartReadOrWrite := TRUE;
		
		//Go to the Next Step
		IF NOT Lynus_Standards.GVL_Bussystems.stDataOfMBRTUMasterKL6xxx[diNrOfMBRTUMasterLine_IN].bMasterIsBusy AND Lynus_Standards.GVL_Bussystems.stDataOfMBRTUMasterKL6xxx[diNrOfMBRTUMasterLine_IN].byErrorWarning = 0 AND timDelay.Q AND 
			diNrOfMBRTUMasterLine_IN = diNrOfMBRTUMasterLine_IN_CP AND byMBAdress_Int = byMBAdress_CP AND NOT timTimeout.Q THEN
				timDelay.IN := FALSE;
					Lynus_Standards.GVL_Bussystems.stDataOfMBRTUMasterKL6xxx[diNrOfMBRTUMasterLine_IN].bSlaveStartReadOrWrite := FALSE;
						iStateModbusRead := 5;	
							wNextModbusStartAdress := wNextModbusStartAdress + 10;	
		END_IF

			//Error on Master, changes on Inputs or Timeout
		 	IF timTimeout.Q OR diNrOfMBRTUMasterLine_IN <> diNrOfMBRTUMasterLine_IN_CP OR byMBAdress_Int <> byMBAdress_CP OR FPErrorMaster.Q THEN 
				iStateModbusError := 300; 
					diNrOfMBRTUMasterLine_IN_CP := diNrOfMBRTUMasterLine_IN; 
						byMBAdress_CP := byMBAdress_Int; 
			END_IF

	5://Read Out Values from Pic 160 of the Sunspec Protocol
		iStateModbus_CP := iStateModbusRead;
		
		wNumberOfMPPT := LIMIT(1,wNumberOfMPPT,6);
			iSFPowerMPPT := LIMIT(-10,iSFPowerMPPT,10);
		
		Lynus_Standards.GVL_Bussystems.stDataOfMBRTUMasterKL6xxx[diNrOfMBRTUMasterLine_IN].eMBRTUReadWriteMode := E_MBRTUMaster_ReadWriteMode.eModbusRTUMaster_ReadRegs;
			Lynus_Standards.GVL_Bussystems.stDataOfMBRTUMasterKL6xxx[diNrOfMBRTUMasterLine_IN].wNumberOfRegister := 20 * wNumberOfMPPT;
				Lynus_Standards.GVL_Bussystems.stDataOfMBRTUMasterKL6xxx[diNrOfMBRTUMasterLine_IN].wModbusRegister := wNextModbusStartAdress;
		
		IF NOT Lynus_Standards.GVL_Bussystems.stDataOfMBRTUMasterKL6xxx[diNrOfMBRTUMasterLine_IN].bMasterIsBusy THEN timDelay.IN := TRUE; END_IF 

		IF wNumberOfMPPT <= 1 THEN
			stDeltaInverterData.arrMPPTPower[2] := 0;
				stDeltaInverterData.arrMPPTPower[3] := 0;
					stDeltaInverterData.arrMPPTPower[4] := 0;
						stDeltaInverterData.arrMPPTPower[5] := 0;
							stDeltaInverterData.arrMPPTPower[6] := 0;
		ELSIF  wNumberOfMPPT = 2 THEN
			stDeltaInverterData.arrMPPTPower[3] := 0;
				stDeltaInverterData.arrMPPTPower[4] := 0;
					stDeltaInverterData.arrMPPTPower[5] := 0;
						stDeltaInverterData.arrMPPTPower[6] := 0;
		ELSIF  wNumberOfMPPT = 3 THEN
			stDeltaInverterData.arrMPPTPower[4] := 0;
				stDeltaInverterData.arrMPPTPower[5] := 0;
					stDeltaInverterData.arrMPPTPower[6] := 0;
		ELSIF  wNumberOfMPPT = 4 THEN
			stDeltaInverterData.arrMPPTPower[5] := 0;
				stDeltaInverterData.arrMPPTPower[6] := 0;	
		ELSIF  wNumberOfMPPT = 5 THEN
			stDeltaInverterData.arrMPPTPower[6] := 0;
		END_IF
		
		//Copy the read out Data
		IF NOT Lynus_Standards.GVL_Bussystems.stDataOfMBRTUMasterKL6xxx[diNrOfMBRTUMasterLine_IN].bMasterIsBusy AND Lynus_Standards.GVL_Bussystems.stDataOfMBRTUMasterKL6xxx[diNrOfMBRTUMasterLine_IN].byErrorWarning = 0 AND timDelay.Q AND diNrOfMBRTUMasterLine_IN = diNrOfMBRTUMasterLine_IN_CP AND byMBAdress_Int = byMBAdress_CP THEN
			//MPPT Power
			FOR wLPPowerMPPT := 1 TO (20 * wNumberOfMPPT) BY 1 DO
				IF wNumberOfMPPT >= 1 AND wLPPowerMPPT = 12 THEN stDeltaInverterData.arrMPPTPower[1] := LREAL_TO_REAL(Lynus_Standards.GVL_Bussystems.stDataOfMBRTUMasterKL6xxx[diNrOfMBRTUMasterLine_IN].arrReadOutData[wLPPowerMPPT] * EXPT(10,iSFPowerMPPT) / 1000);
				ELSIF wNumberOfMPPT >= 2 AND wLPPowerMPPT = 32 THEN stDeltaInverterData.arrMPPTPower[2] := LREAL_TO_REAL(Lynus_Standards.GVL_Bussystems.stDataOfMBRTUMasterKL6xxx[diNrOfMBRTUMasterLine_IN].arrReadOutData[wLPPowerMPPT] * EXPT(10,iSFPowerMPPT) / 1000);
				ELSIF wNumberOfMPPT >= 3 AND wLPPowerMPPT = 52 THEN stDeltaInverterData.arrMPPTPower[3] := LREAL_TO_REAL(Lynus_Standards.GVL_Bussystems.stDataOfMBRTUMasterKL6xxx[diNrOfMBRTUMasterLine_IN].arrReadOutData[wLPPowerMPPT] * EXPT(10,iSFPowerMPPT) / 1000);
				ELSIF wNumberOfMPPT >= 4 AND wLPPowerMPPT = 72 THEN stDeltaInverterData.arrMPPTPower[4] := LREAL_TO_REAL(Lynus_Standards.GVL_Bussystems.stDataOfMBRTUMasterKL6xxx[diNrOfMBRTUMasterLine_IN].arrReadOutData[wLPPowerMPPT] * EXPT(10,iSFPowerMPPT) / 1000);
				ELSIF wNumberOfMPPT >= 5 AND wLPPowerMPPT = 92 THEN stDeltaInverterData.arrMPPTPower[5] := LREAL_TO_REAL(Lynus_Standards.GVL_Bussystems.stDataOfMBRTUMasterKL6xxx[diNrOfMBRTUMasterLine_IN].arrReadOutData[wLPPowerMPPT] * EXPT(10,iSFPowerMPPT) / 1000);
				ELSIF wNumberOfMPPT >= 6 AND wLPPowerMPPT = 112 THEN stDeltaInverterData.arrMPPTPower[6] := LREAL_TO_REAL(Lynus_Standards.GVL_Bussystems.stDataOfMBRTUMasterKL6xxx[diNrOfMBRTUMasterLine_IN].arrReadOutData[wLPPowerMPPT] * EXPT(10,iSFPowerMPPT) / 1000);
				END_IF     
			END_FOR 
		END_IF     				
		
		//Total DC Power
		stDeltaInverterData.rTotalMPPTPower := 0;
			FOR wLPPowerMPPT := 1 TO 6 BY 1 DO
				stDeltaInverterData.rTotalMPPTPower := stDeltaInverterData.rTotalMPPTPower + stDeltaInverterData.arrMPPTPower[wLPPowerMPPT];
			END_FOR
			
		//Send the Read or Write Command to the Master
		Lynus_Standards.GVL_Bussystems.stDataOfMBRTUMasterKL6xxx[diNrOfMBRTUMasterLine_IN].bSlaveStartReadOrWrite := TRUE;
		
		//Go to the Next Step
		IF NOT Lynus_Standards.GVL_Bussystems.stDataOfMBRTUMasterKL6xxx[diNrOfMBRTUMasterLine_IN].bMasterIsBusy AND Lynus_Standards.GVL_Bussystems.stDataOfMBRTUMasterKL6xxx[diNrOfMBRTUMasterLine_IN].byErrorWarning = 0 AND timDelay.Q AND 
			diNrOfMBRTUMasterLine_IN = diNrOfMBRTUMasterLine_IN_CP AND byMBAdress_Int = byMBAdress_CP AND NOT timTimeout.Q THEN
				timDelay.IN := FALSE;
					Lynus_Standards.GVL_Bussystems.stDataOfMBRTUMasterKL6xxx[diNrOfMBRTUMasterLine_IN].bSlaveStartReadOrWrite := FALSE;
						iStateModbusRead := 6;
							lrRestNextAdress := 0;		
			//Calculate next Modbus Start Adress for Pic 401
			wNextModbusStartAdress := wNextModbusStartAdress - 10;
				wNextModbusStartAdress := wNextModbusStartAdress + wNumberOfInputs + 2;
					lrRestNextAdress := FRAC(WORD_TO_REAL(wNextModbusStartAdress) / 2);	
						//If it ends with an odd number, the next PIC starts with an even address
						IF lrRestNextAdress <> 0 THEN wNextModbusStartAdress := wNextModbusStartAdress + 1; END_IF
		END_IF

			//Error on Master, changes on Inputs or Timeout
		 	IF timTimeout.Q OR diNrOfMBRTUMasterLine_IN <> diNrOfMBRTUMasterLine_IN_CP OR byMBAdress_Int <> byMBAdress_CP OR FPErrorMaster.Q THEN 
				iStateModbusError := 300; 
					diNrOfMBRTUMasterLine_IN_CP := diNrOfMBRTUMasterLine_IN; 
						byMBAdress_CP := byMBAdress_Int; 
			END_IF
	
	6://Read Out Values from Pic 401 to Start Adress for Vendor 64062 of the Sunspec Protocoll	
		iStateModbus_CP := iStateModbusRead;
		
		Lynus_Standards.GVL_Bussystems.stDataOfMBRTUMasterKL6xxx[diNrOfMBRTUMasterLine_IN].eMBRTUReadWriteMode := E_MBRTUMaster_ReadWriteMode.eModbusRTUMaster_ReadRegs;
			Lynus_Standards.GVL_Bussystems.stDataOfMBRTUMasterKL6xxx[diNrOfMBRTUMasterLine_IN].wNumberOfRegister := 2;
				Lynus_Standards.GVL_Bussystems.stDataOfMBRTUMasterKL6xxx[diNrOfMBRTUMasterLine_IN].wModbusRegister := wNextModbusStartAdress;
		
		IF NOT Lynus_Standards.GVL_Bussystems.stDataOfMBRTUMasterKL6xxx[diNrOfMBRTUMasterLine_IN].bMasterIsBusy THEN timDelay.IN := TRUE; END_IF 

		//Copy the read out Data
		IF NOT Lynus_Standards.GVL_Bussystems.stDataOfMBRTUMasterKL6xxx[diNrOfMBRTUMasterLine_IN].bMasterIsBusy AND Lynus_Standards.GVL_Bussystems.stDataOfMBRTUMasterKL6xxx[diNrOfMBRTUMasterLine_IN].byErrorWarning = 0 AND timDelay.Q AND diNrOfMBRTUMasterLine_IN = diNrOfMBRTUMasterLine_IN_CP AND byMBAdress_Int = byMBAdress_CP THEN
			//PIC ID
			wPicID := Lynus_Standards.GVL_Bussystems.stDataOfMBRTUMasterKL6xxx[diNrOfMBRTUMasterLine_IN].arrReadOutData[1];
			//Number of Inputs
			wNumberOfInputs := Lynus_Standards.GVL_Bussystems.stDataOfMBRTUMasterKL6xxx[diNrOfMBRTUMasterLine_IN].arrReadOutData[2];
		END_IF     					
		
		//Send the Read or Write Command to the Master
		Lynus_Standards.GVL_Bussystems.stDataOfMBRTUMasterKL6xxx[diNrOfMBRTUMasterLine_IN].bSlaveStartReadOrWrite := TRUE;
		
		//Go to the Next Step
		IF NOT Lynus_Standards.GVL_Bussystems.stDataOfMBRTUMasterKL6xxx[diNrOfMBRTUMasterLine_IN].bMasterIsBusy AND Lynus_Standards.GVL_Bussystems.stDataOfMBRTUMasterKL6xxx[diNrOfMBRTUMasterLine_IN].byErrorWarning = 0 AND timDelay.Q AND 
			diNrOfMBRTUMasterLine_IN = diNrOfMBRTUMasterLine_IN_CP AND byMBAdress_Int = byMBAdress_CP AND NOT timTimeout.Q THEN
				timDelay.IN := FALSE;
					Lynus_Standards.GVL_Bussystems.stDataOfMBRTUMasterKL6xxx[diNrOfMBRTUMasterLine_IN].bSlaveStartReadOrWrite := FALSE;
						iStateModbusRead := 7;	
							lrRestNextAdress := 0;
			//Calculate next Modbus Start Adress
			wNextModbusStartAdress := wNextModbusStartAdress + wNumberOfInputs + 2;
				lrRestNextAdress := FRAC(WORD_TO_REAL(wNextModbusStartAdress) / 2);	
					//If it ends with an odd number, the next PIC starts with an even address
					IF lrRestNextAdress <> 0 THEN wNextModbusStartAdress := wNextModbusStartAdress + 1; END_IF 
		END_IF

			//Error on Master, changes on Inputs or Timeout
		 	IF timTimeout.Q OR diNrOfMBRTUMasterLine_IN <> diNrOfMBRTUMasterLine_IN_CP OR byMBAdress_Int <> byMBAdress_CP OR FPErrorMaster.Q THEN 
				iStateModbusError := 300; 
					diNrOfMBRTUMasterLine_IN_CP := diNrOfMBRTUMasterLine_IN; 
						byMBAdress_CP := byMBAdress_Int; 
			END_IF
	
	7://Check the PIC ID
		iStateModbus_CP := iStateModbusRead;
		
		IF wPicID < 64062 THEN
			//Back to Step 6
			iStateModbusRead := 6;
		ELSE
			//next Step with values
			iStateModbusRead := 8;
				//Calculate next Modbus Start Adress for next Pic or Vendor
				wNextModbusStartAdress := wNextModbusStartAdress - wNumberOfInputs - 2;
		END_IF		
			
	8://Read Out Values from Pic Vendor 64062 of the Sunspec Protocol (Register wNextModbusStartAdress + 2)		
		iStateModbus_CP := iStateModbusRead;
		
		Lynus_Standards.GVL_Bussystems.stDataOfMBRTUMasterKL6xxx[diNrOfMBRTUMasterLine_IN].eMBRTUReadWriteMode := E_MBRTUMaster_ReadWriteMode.eModbusRTUMaster_ReadRegs;
			Lynus_Standards.GVL_Bussystems.stDataOfMBRTUMasterKL6xxx[diNrOfMBRTUMasterLine_IN].wNumberOfRegister := 16;
				Lynus_Standards.GVL_Bussystems.stDataOfMBRTUMasterKL6xxx[diNrOfMBRTUMasterLine_IN].wModbusRegister := wNextModbusStartAdress + 2;
		
		IF NOT Lynus_Standards.GVL_Bussystems.stDataOfMBRTUMasterKL6xxx[diNrOfMBRTUMasterLine_IN].bMasterIsBusy THEN timDelay.IN := TRUE; END_IF 

		//Copy the read out Data
		IF NOT Lynus_Standards.GVL_Bussystems.stDataOfMBRTUMasterKL6xxx[diNrOfMBRTUMasterLine_IN].bMasterIsBusy AND Lynus_Standards.GVL_Bussystems.stDataOfMBRTUMasterKL6xxx[diNrOfMBRTUMasterLine_IN].byErrorWarning = 0 AND timDelay.Q AND diNrOfMBRTUMasterLine_IN = diNrOfMBRTUMasterLine_IN_CP AND byMBAdress_Int = byMBAdress_CP THEN
			//Faults
			FOR byLPVendor64062 := 1 TO 8 BY 1 DO 
				stDeltaInverterData.arrCurrentFault[byLPVendor64062] := Lynus_Standards.GVL_Bussystems.stDataOfMBRTUMasterKL6xxx[diNrOfMBRTUMasterLine_IN].arrReadOutData[byLPVendor64062];
			END_FOR
			//Error
			FOR byLPVendor64062 := 9 TO 13 BY 1 DO 
				stDeltaInverterData.arrCurrentError[byLPVendor64062 - 8] := Lynus_Standards.GVL_Bussystems.stDataOfMBRTUMasterKL6xxx[diNrOfMBRTUMasterLine_IN].arrReadOutData[byLPVendor64062];
			END_FOR
			//Warning
			FOR byLPVendor64062 := 14 TO 16 BY 1 DO 
				stDeltaInverterData.arrCurrentError[byLPVendor64062 - 13] := Lynus_Standards.GVL_Bussystems.stDataOfMBRTUMasterKL6xxx[diNrOfMBRTUMasterLine_IN].arrReadOutData[byLPVendor64062];
			END_FOR
		END_IF     				
		
		//Send the Read or Write Command to the Master
		Lynus_Standards.GVL_Bussystems.stDataOfMBRTUMasterKL6xxx[diNrOfMBRTUMasterLine_IN].bSlaveStartReadOrWrite := TRUE;
		
		//Go to the Next Step
		IF NOT Lynus_Standards.GVL_Bussystems.stDataOfMBRTUMasterKL6xxx[diNrOfMBRTUMasterLine_IN].bMasterIsBusy AND Lynus_Standards.GVL_Bussystems.stDataOfMBRTUMasterKL6xxx[diNrOfMBRTUMasterLine_IN].byErrorWarning = 0 AND timDelay.Q AND 
			diNrOfMBRTUMasterLine_IN = diNrOfMBRTUMasterLine_IN_CP AND byMBAdress_Int = byMBAdress_CP AND NOT timTimeout.Q THEN
				timDelay.IN := FALSE;
					Lynus_Standards.GVL_Bussystems.stDataOfMBRTUMasterKL6xxx[diNrOfMBRTUMasterLine_IN].bSlaveStartReadOrWrite := FALSE;
						Lynus_Standards.GVL_Bussystems.stDataOfMBRTUMasterKL6xxx[diNrOfMBRTUMasterLine_IN].bReadWriteIsDone := TRUE;
							iStateModbusRead := 0;		
		END_IF

			//Error on Master, changes on Inputs or Timeout
		 	IF timTimeout.Q OR diNrOfMBRTUMasterLine_IN <> diNrOfMBRTUMasterLine_IN_CP OR byMBAdress_Int <> byMBAdress_CP OR FPErrorMaster.Q THEN 
				iStateModbusError := 300; 
					diNrOfMBRTUMasterLine_IN_CP := diNrOfMBRTUMasterLine_IN; 
						byMBAdress_CP := byMBAdress_Int; 
			END_IF
	
END_CASE

(*------------------------------------------------------------------Error and Warning----------------------------------------------------------------------------*)	

bErrorInverter := FALSE;
	bWarningInverter := FALSE;
		FOR byLPVendor64062 := 1 TO 8 BY 1 DO 
			IF stDeltaInverterData.arrCurrentFault[byLPVendor64062] <> 0 AND stDeltaInverterData.eOperatingState = eDeltaOperatingState.eFault THEN bErrorInverter := TRUE; END_IF
		END_FOR
			FOR byLPVendor64062 := 1 TO 5 BY 1 DO 
				IF stDeltaInverterData.arrCurrentError[byLPVendor64062] <> 0 AND stDeltaInverterData.eEvent1 = eDeltaEvent.eOtherAlarm THEN bErrorInverter := TRUE; END_IF
			END_FOR
				FOR byLPVendor64062 := 1 TO 3 BY 1 DO 
					IF stDeltaInverterData.arrCurrentWarning[byLPVendor64062] <> 0 AND stDeltaInverterData.eEvent1 = eDeltaEvent.eOtherWarning THEN bWarningInverter := TRUE; END_IF
				END_FOR
					IF stDeltaInverterData.eOperatingState = eDeltaOperatingState.eFault THEN bErrorInverter := TRUE; END_IF
						IF stDeltaInverterData.eEvent1 <> eDeltaEvent.eNoInfo THEN bErrorInverter := TRUE; END_IF    

IF timDissableFunctions.Q OR bWarningInverter THEN fbElMeter.bWarning := TRUE; ELSE fbElMeter.bWarning := FALSE; fbElMeter.iWarningCode := 0; END_IF   
	IF Lynus_Standards.GVL_Energy.stNumberOfDevices.diNumberOfElectricMeters > Constants_Energy.diMaxNumberOfElectricMeters OR bErrorInverter OR Lynus_Standards.GVL_Bussystems.stDataOfMBRTUMasterKL6xxx[diNrOfMBRTUMasterLine_IN].byErrorWarning = 2 OR timTimeout.Q THEN 
		fbElMeter.bError := TRUE;
	ELSE 
		fbElMeter.bError := FALSE;
			fbElMeter.iErrorCode := 0;
	END_IF

IF timDissableFunctions.Q THEN fbElMeter.iWarningCode := 0;
ELSIF bWarningInverter THEN fbElMeter.iWarningCode := 1;
END_IF    	
	
IF Lynus_Standards.GVL_Energy.stNumberOfDevices.diNumberOfElectricMeters > Constants_Energy.diMaxNumberOfElectricMeters THEN fbElMeter.iErrorCode := 1; END_IF
	IF Lynus_Standards.GVL_Bussystems.stDataOfMBRTUMasterKL6xxx[diNrOfMBRTUMasterLine_IN].byErrorWarning = 2 OR bErrorInverter OR timTimeout.Q THEN fbElMeter.iErrorCode := 0; END_IF   

(*------------------------------------------------------------------Logic----------------------------------------------------------------------------*)

//Read Out Data done for EM Function
IF iStateModbusRead <> 1 THEN fbElMeter.bReadOutDataDone := TRUE; ELSE fbElMeter.bReadOutDataDone := FALSE; END_IF

//Function block for meter data
fbElMeter(
	bEnable:= bEnable AND NOT timDissableFunctions.Q, 
	bError:= , 
	bEnableReadOutFunction:= FALSE, 
	bWriteWithDelay:= TRUE,
	bPowerDataInvers:= FALSE, 
	bReadOutDataDone:= ,
	iTimeReadOutInterval:= , 
	iErrorCode:= , 
	iWarningCode:= , 
	lrTotalCounterEnergy_Consumption:= 0, 
	lrTotalCounterEnergy_Production:= , 
	lrCounterEnergyT1_Consumption:= 0, 
	lrCounterEnergyT2_Consumption:= 0, 
	lrCounterEnergyT1_Production:= , 
	lrCounterEnergyT2_Production:= 0, 
	lrCurrentL1:= , 
	lrVoltageL1N:= , 
	lrVoltageL1L2:= , 
	lrPowerL1:= 0, 
	lrCurrentL2:= , 
	lrVoltageL2N:= , 
	lrVoltageL2L3:= , 
	lrPowerL2:= 0, 
	lrCurrentL3:= , 
	lrVoltageL3N:= , 
	lrVoltageL3L1:= , 
	lrPowerL3:= 0, 
	lrPowerTotal:= , 
	lrFrequency:= , 
	lrReactivePowerTotal:= , 
	lrApparentPowerTotal:= , 
	tTimDelayOutput:= T#5S, 
	stDataEMOutPower=> , 
	stDataEMOutPowerDelay=> stDataEMPower_PV, 
	stDataEMOutCounter=> ,
	stDataEMOutCounterDelay=> stDataEMCounter_PV, 
	bReadOutMeter=> );
	
(*------------------------------------------------------------------------------------------State Machine Error---------------------------------------------------------------------------------------------*)	

CASE iStateModbusError OF
	
	300://Error
		iStateModbus_CP := iStateModbusError;
			timDelay.IN := FALSE;
				Lynus_Standards.GVL_Bussystems.stDataOfMBRTUMasterKL6xxx[diNrOfMBRTUMasterLine_IN].bSlaveStartReadOrWrite := FALSE;
					//Restart from new with the Read out part after an Error
					iStateModbusRead := 0;	
						iStateModbusError := 0;
END_CASE

(*------------------------------------------------------------------------------------------Device Type for MB RTU Master---------------------------------------------------------------------------------------------*)	

//Send the Device Type to the Master that he can configure the Termial with the right credentials
Lynus_Standards.GVL_Bussystems.stDataOfMBRTUMasterKL6xxx[diNrOfMBRTUMasterLine_IN].eMBRTUDeviceType := E_MBRTUMaster_DeviceType.ePV_DeltaSunspec;

(*-----------------------------------------------------------Handle data to Global structure for Electric Meter system and Modbus RTU Communication-----------------------------------------------------------------*)

CASE iStateGVLData OF
	
	0://Init Step
		byWaitInStep := 0;
			arrCounterForGVL[1] := 1; arrCounterForGVL[2] := 1;
	
	1://Wait for 4 Steps before clean al Data on GVL
		byWaitInStep := byWaitInStep + 1;
			IF byWaitInStep >= 4 AND fbNumberDevice.bNumberIsCalculatet THEN iStateGVLData := 2; END_IF
				//To much Devices, back to the Init step
				IF byWaitInStep >= 4 AND NOT fbNumberDevice.bNumberIsCalculatet THEN iStateGVLData := 0; END_IF	
			
	2://Clear all Data in GVL
		Lynus_Standards.GVL_Energy.stDataElectricMeters[arrCounterForGVL[1]].bEnabled := FALSE;	
			Lynus_Standards.GVL_Energy.stDataElectricMeters[arrCounterForGVL[1]].byErrorWarning := 0;
				Lynus_Standards.GVL_Energy.stDataElectricMeters[arrCounterForGVL[1]].lrCounterEnergyT1_Consumption := 0;
					Lynus_Standards.GVL_Energy.stDataElectricMeters[arrCounterForGVL[1]].lrCounterEnergyT1_Production := 0;
						Lynus_Standards.GVL_Energy.stDataElectricMeters[arrCounterForGVL[1]].lrCounterEnergyT2_Consumption := 0;
							Lynus_Standards.GVL_Energy.stDataElectricMeters[arrCounterForGVL[1]].lrCounterEnergyT2_Production := 0;
								Lynus_Standards.GVL_Energy.stDataElectricMeters[arrCounterForGVL[1]].lrPower := 0;
									Lynus_Standards.GVL_Energy.stDataElectricMeters[arrCounterForGVL[1]].lrPowerConsumption := 0;
										Lynus_Standards.GVL_Energy.stDataElectricMeters[arrCounterForGVL[1]].lrPowerConsumption := 0;
											Lynus_Standards.GVL_Energy.stDataElectricMeters[arrCounterForGVL[1]].lrPowerProduction := 0;
												Lynus_Standards.GVL_Energy.stDataElectricMeters[arrCounterForGVL[1]].lrTotalCounterEnergy_Consumption := 0;
													Lynus_Standards.GVL_Energy.stDataElectricMeters[arrCounterForGVL[1]].lrTotalCounterEnergy_Production := 0;
		
			//Reset this Part here and not in the RTU Master because on top we write then the New Adess in the List. So in the Master we delete only the GVL after a online change what set the Master by himself
			Lynus_Standards.GVL_Bussystems.stDataOfMBRTUMasterKL6xxx[arrCounterForGVL[2]].arrAllModbusSlaveAdresses := arrDefaultModbusAdress;
				Lynus_Standards.GVL_Bussystems.stDataOfMBRTUMasterKL6xxx[arrCounterForGVL[2]].arrReadOutData := arrDefaultReadWrite;
					Lynus_Standards.GVL_Bussystems.stDataOfMBRTUMasterKL6xxx[arrCounterForGVL[2]].arrWriteOutData := arrDefaultReadWrite;
						Lynus_Standards.GVL_Bussystems.stDataOfMBRTUMasterKL6xxx[arrCounterForGVL[2]].bSlaveStartReadOrWrite := FALSE;
							Lynus_Standards.GVL_Bussystems.stDataOfMBRTUMasterKL6xxx[arrCounterForGVL[2]].eMBRTUDeviceType := E_MBRTUMaster_DeviceType.eNoModbusRTUDevice;
								Lynus_Standards.GVL_Bussystems.stDataOfMBRTUMasterKL6xxx[arrCounterForGVL[2]].eMBRTUReadWriteMode := E_MBRTUMaster_ReadWriteMode.eModbusRTUMaster_NoMode;
									Lynus_Standards.GVL_Bussystems.stDataOfMBRTUMasterKL6xxx[arrCounterForGVL[2]].wModbusRegister := 0;
										Lynus_Standards.GVL_Bussystems.stDataOfMBRTUMasterKL6xxx[arrCounterForGVL[2]].wNumberOfRegister := 0;			
		
			//Counter for MB RTU Master
			arrCounterForGVL[2] := arrCounterForGVL[2] + 1;
				arrCounterForGVL[2] := LIMIT(0,arrCounterForGVL[2],Constants_Bussystems.diMaxNumberOfMBRTUMasterKL6xxx);
			//Counter for EM
			arrCounterForGVL[1] := arrCounterForGVL[1] + 1;
				arrCounterForGVL[1] := LIMIT(0,arrCounterForGVL[1],Constants_Energy.diMaxNumberOfElectricMeters);
					//Back to the init step
					IF arrCounterForGVL[1] >= Constants_Energy.diMaxNumberOfElectricMeters AND arrCounterForGVL[2] >= Constants_Bussystems.diMaxNumberOfMBRTUMasterKL6xxx THEN iStateGVLData := 0; END_IF

END_CASE 	 

IF diNrOfEM_OUT_PV > 0 AND fbNumberDevice.bNumberIsCalculatet THEN
	Lynus_Standards.GVL_Energy.stDataElectricMeters[diNrOfEM_OUT_PV].bEnabled := fbElMeter.stDataEMOutPower.bEnabled;
		Lynus_Standards.GVL_Energy.stDataElectricMeters[diNrOfEM_OUT_PV].byErrorWarning := fbElMeter.stDataEMOutPower.byErrorWarning;
			Lynus_Standards.GVL_Energy.stDataElectricMeters[diNrOfEM_OUT_PV].lrCounterEnergyT1_Consumption := fbElMeter.stDataEMOutCounter.lrCounterEnergyT1_Consumption;
				Lynus_Standards.GVL_Energy.stDataElectricMeters[diNrOfEM_OUT_PV].lrCounterEnergyT1_Production := fbElMeter.stDataEMOutCounter.lrCounterEnergyT1_Production;
					Lynus_Standards.GVL_Energy.stDataElectricMeters[diNrOfEM_OUT_PV].lrCounterEnergyT2_Consumption := fbElMeter.stDataEMOutCounter.lrCounterEnergyT2_Consumption;
						Lynus_Standards.GVL_Energy.stDataElectricMeters[diNrOfEM_OUT_PV].lrCounterEnergyT2_Production := fbElMeter.stDataEMOutCounter.lrCounterEnergyT2_Production;		
							Lynus_Standards.GVL_Energy.stDataElectricMeters[diNrOfEM_OUT_PV].lrPower := fbElMeter.stDataEMOutPower.lrPowerTotal;
								Lynus_Standards.GVL_Energy.stDataElectricMeters[diNrOfEM_OUT_PV].lrPowerConsumption := fbElMeter.stDataEMOutPower.lrPowerConsumption;
									Lynus_Standards.GVL_Energy.stDataElectricMeters[diNrOfEM_OUT_PV].lrPowerProduction := fbElMeter.stDataEMOutPower.lrPowerProduction;
										Lynus_Standards.GVL_Energy.stDataElectricMeters[diNrOfEM_OUT_PV].lrTotalCounterEnergy_Consumption := fbElMeter.stDataEMOutCounter.lrTotalCounterEnergy_Consumption;
											Lynus_Standards.GVL_Energy.stDataElectricMeters[diNrOfEM_OUT_PV].lrTotalCounterEnergy_Production := fbElMeter.stDataEMOutCounter.lrTotalCounterEnergy_Production;
END_IF

(*----------------------------------------------------------Save persistent data----------------------------------------------------------------*)

arrPD[1](lrValue:= BOOL_TO_LREAL(bEnable), bEventBasedActive=> );
arrPD[2](lrValue:= BYTE_TO_LREAL(byMBAdress), bEventBasedActive=> );
arrPD[3](lrValue:= DINT_TO_LREAL(diNrOfMBRTUMasterLine_IN), bEventBasedActive=> );
arrPD[4](lrValue:= BYTE_TO_LREAL(byMBAdress_ForChange), bEventBasedActive=> );
arrPD[5](lrValue:= BYTE_TO_LREAL(byMBAdress_Int), bEventBasedActive=> );

END_FUNCTION_BLOCK

// ---- FBs/Modbus RTU Master/FB_KL6xxx_ModbusRTU_22B_Master.TcPOU
FUNCTION_BLOCK FB_KL6xxx_ModbusRTU_22B_Master
VAR_INPUT
	bConfigTerminal							: BOOL;																		//Possibility to configure the Terminal manually (Its only possible when the Terminal is not configured successfully)
	uiKBusState_IN							: UINT;																		//K-Bus State from the K-Bus Box on wich the Terminal is connected. (Connect with FB_K_Bus_state)
END_VAR
VAR_OUTPUT
	bBusy									: BOOL;																		//Function is Busy
	byErrorWarning							: BYTE;																		//Error Warning State
	byActualAdressInUse						: BYTE;																		//Actual Modbus Adress in Use
	diNrOfMBRTUMasterLine_OUT				: DINT;																		//Active Number from the RTU Master Function for using on other functions
	eMessageMBRTUMaster						: E_Message_MBRTUMaster;													//Message from the RTU Master Function
END_VAR				
VAR_OUTPUT PERSISTENT
	bTerminalIsConfigured					: BOOL;																		//Its True when the configuration is successfully
END_VAR
VAR		
	{attribute 'hide'}
	fbKL6xxxConfig							: KL6configuration;															//FB KL6xxx to config the terminal
	fbmodbusmaster							: ModbusRtuMaster_KL6x22B;													//FB Modbus RTU
	{attribute 'hide'}
	fbmodbusmaster_Init						: ModbusRtuMaster_KL6x22B;													//FB Modbus RTU Master for workaroud regarding the internal Beckhoff problem in this function
	{attribute 'hide'}
	fbNumberDevice							: FB_NumberOfDevice;														//Function block to calcualte the number of the Device	
	{attribute 'hide'}
	fbModbusRTUMessage						: FB_MBRTUMaster_Messages;													//Modbus RTU Messages	
	{attribute 'hide'}
	FPConfigManual							: R_TRIG;																	//Internal positive Edge
	{attribute 'hide'}
	FPConfigAuto							: R_TRIG;																	//Internal positive Edge
	{attribute 'hide'}
	FPProcessCompleted						: R_TRIG;																	//Internal positive Edge
	{attribute 'hide'}
	FPError									: R_TRIG;																	//Internal positive Edge
	{attribute 'hide'}
	FPErrorIsActive							: R_TRIG;																	//Internal positive Edge
	{attribute 'hide'}
	FNInitSmall								: F_TRIG;																	//Internal negative Edge
	{attribute 'hide'}
	FNBusy									: F_TRIG;																	//Internal negative Edge
	{attribute 'hide'}
	timInit									: TON;																		//Delay to start the Terminal Configuration after the start from the plc
	{attribute 'hide'}
	timTimout								: TON;																		//Timer Timout to go on next Modbus Adress when the Ack is not set back to False
	{attribute 'hide'}
	timDissableFunctions					: TON;																		//Timer to dissable the Function after Lynus_Standards.Constants_General.tTimeDissableLynusFunctions Days without connection to the Lynus Cloud
	{attribute 'hide'}
	timResetConnectionOnGVL					: TON;																		//Timer to try reset the connection Flag on the GVL. (When somebody delete the Connection Function and make only a onlinechange)
	{attribute 'hide'}
	arrPD									: ARRAY[1..2] OF FB_PersistentData_Number;									//Function to save persistent data
	{attribute 'hide'}
	bTakeActualAdress						: BOOL;																		//True if the Current address is to be used
	{attribute 'hide'}
	bAdressHasChanged						: BOOL;																		//True if the Adress has changed
	{attribute 'hide'}
	bErrorIsActive							: BOOL;																		//True if a Error is happend. False after the next successfully read or write command
	{attribute 'hide'}
	bStopReadWrite							: BOOL;																		//Stop Function because Modbus Adress has chaged
	{attribute 'hide'}
	byLPSmallestAdress						: BYTE;																		//Loop to find out the smallest Modbus Adress
	{attribute 'hide'}
	byLPBiggestAdress						: BYTE;																		//Loop to find out the biggest Modbus Adress
	{attribute 'hide'}
	byLPActualAdress						: BYTE;																		//Loop to find out the next actuall adress
	{attribute 'hide'}
	byLPNumbersOfTotalSlaves				: BYTE;																		//Loop to find out the number of total Modbus Slaves
	{attribute 'hide'}
	bySmallestAdress						: BYTE;																		//Smallest Modbus Adress
	{attribute 'hide'}
	byBiggestAdress							: BYTE;																		//Biggest Modbus Adress
	{attribute 'hide'}
	byActualAdressInUse_CP					: BYTE;																		//Actual Modbus Adress in Use to compare it with the old one
	{attribute 'hide'}
	byNumberOfTotalSlaves					: BYTE;																		//Number of all Modbus Slaves
	{attribute 'hide'}
	byWaitInStep							: BYTE;																		//Wait in Step before start to clean data on PLC
	{attribute 'hide'}
	byLPMBAdress							: BYTE;																		//Loop for manage new Modbus Adress List after a change
	{attribute 'hide'}
	bySearchMBAdress						: BYTE;																		//Search Modbus Adress after change
	{attribute 'hide'}
	byPosInArrayMBAdress					: BYTE;																		//Save new Range from Modbus adress in the Array after a change
	{attribute 'hide'}
	iStateGVLData							: INT;																		//State machine to handle the data on the GVL
	{attribute 'hide'}
	iStateSetMBAdress						: INT;																		//State machin eto order the Modbus Adress after a change
	{attribute 'hide'}
	diCounterForGVL							: DINT;																		//Counter to clean old data on GVL
	{attribute 'hide'}
	arrRead									: ARRAY[1..Constants_Bussystems.wQuantityOfRegistersMBRTUMaster] OF WORD;	//Puffer for read out data
	{attribute 'hide'}
	arrMBAdress								: ARRAY[1..247] OF BYTE;													//Array with the actual Modbus Adress Config
END_VAR
VAR PERSISTENT
	{attribute 'conditionalshow'}
	eDeviceType								: E_MBRTUMaster_DeviceType;													//Device Type on witch the Terminal is configured
END_VAR

//Creator : Kai Ebensperger
//Company : Lynus AG
//Date : 08.07.2021
//Version : 1.0.0.0

//With this FB a serial 22 byte terminal can be configured and data can be sent/received via Modbus RTU.
//Only devices of the same type may be operated on the same master (because its not good to write to much new configurations on the terminal).
//The 1 slave that is called before the master FB in the PLC code configures the terminal
//The block must be called in a task of 5MS
//The system works according to the Master Slave principle
//Multiple communication is not possible in RTU principle

//NOTE for diNr.....Designation => 
//_IN = Here Data come in from other Functions or go out to other functions about the GVL
//_OUT = Here Data go out to other functions about the GVL

(*-------------------------------------------------------------Calcualte the number of RTU Master---------------------------------------------------------------*)

fbNumberDevice(
	diActualNumberOfDevices:= Lynus_Standards.GVL_Bussystems.diNumberOfMBRTUMasters, 
	diMaxNumberOfDevices:= Constants_Bussystems.diMaxNumberOfMBRTUMasterKL6xxx, 
	udiCounterOnlineChange:= TwinCAT_SystemInfoVarList._AppInfo.OnlineChangeCnt, 
	bNumberIsCalculatet=> , 
	bFPNumberIsCalculatet=> , 
	bOnlineChange=> , 
	diNumberForThisDevice=> diNrOfMBRTUMasterLine_OUT, 
	diNumberOfTotalDevices=> );

//Write new Numer on GVL
IF fbNumberDevice.bFPNumberIsCalculatet THEN
	Lynus_Standards.GVL_Bussystems.diNumberOfMBRTUMasters := fbNumberDevice.diNumberOfTotalDevices;	
END_IF 

//Delete old Number on GVL
IF fbNumberDevice.bOnlineChange THEN 
	Lynus_Standards.GVL_Bussystems.diNumberOfMBRTUMasters := diNrOfMBRTUMasterLine_OUT;	
		iStateGVLData := 1; 
END_IF	
	
(*-------------------------------------------------------------Service from Backend is ready and check the connection to backen for dissabel/enable Function---------------------------------------------------------------*)

//Try to reset the variable for connection on the GVL. When all is normal then the Lynus Mqtt connection function set this variable to true in the next cycle
//When we have no connection to the backend then after Lynus_Standards.Constants_General.tTimeDissableLynusFunctions days the Function is dissabled with all of his functionalities
timResetConnectionOnGVL(IN:= NOT timResetConnectionOnGVL.Q, PT:= T#1H, Q=> , ET=> );
	IF timResetConnectionOnGVL.Q THEN Lynus_Standards.GVL_Communicator.bStateConnectionToEnableFunctions := FALSE; END_IF
		IF NOT Lynus_Standards.GVL_Communicator.bStateConnectionToEnableFunctions THEN timDissableFunctions.IN := TRUE; ELSE timDissableFunctions.IN := FALSE; END_IF  
			timDissableFunctions(IN:= , PT:= Lynus_Standards.Constants_General.tTimeDissableLynusFunctions, Q=> , ET=> );

(*------------------------------------------------------------------Configuration----------------------------------------------------------------------------*)
			
//Configurate the seriall Terminal
//The configuration is depending what Slave is connected to the terminal
timInit(IN:= Lynus_Standards.GVL_Bussystems.stDataOfMBRTUMasterKL6xxx[diNrOfMBRTUMasterLine_OUT].eMBRTUDeviceType <> E_MBRTUMaster_DeviceType.eNoModbusRTUDevice AND uiKBusState_IN = 0, PT:=T#500MS, Q=> , ET=> );

IF Lynus_Standards.GVL_Bussystems.stDataOfMBRTUMasterKL6xxx[diNrOfMBRTUMasterLine_OUT].eMBRTUDeviceType <> eDeviceType AND timInit.Q THEN
	FPConfigAuto.CLK := TRUE;
		eDeviceType := Lynus_Standards.GVL_Bussystems.stDataOfMBRTUMasterKL6xxx[diNrOfMBRTUMasterLine_OUT].eMBRTUDeviceType;
ELSE
	FPConfigAuto.CLK := FALSE;
END_IF 	 

FPConfigAuto(CLK:= , Q=> );

//Configuration from the Terminal by the Slave Type
IF Lynus_Standards.GVL_Bussystems.stDataOfMBRTUMasterKL6xxx[diNrOfMBRTUMasterLine_OUT].eMBRTUDeviceType = E_MBRTUMaster_DeviceType.ePilotPMAC201_HW THEN
	//Pilot PMAC201 HW Energymessurement Device
	fbKL6xxxConfig.Mode := SERIALLINEMODE_KL6_22B_STANDARD;
	fbKL6xxxConfig.Baudrate := 38400;
	fbKL6xxxConfig.NoDatabits := 8;
	fbKL6xxxConfig.Parity := PARITY_NONE;
	fbKL6xxxConfig.Stopbits := 1;
	fbKL6xxxConfig.Handshake := RS485_HALFDUPLEX;
	fbKL6xxxConfig.ContinousMode := FALSE;
	//Timout	
	timTimout.PT := T#2S;
	fbmodbusmaster.Timeout := T#2S;
ELSIF Lynus_Standards.GVL_Bussystems.stDataOfMBRTUMasterKL6xxx[diNrOfMBRTUMasterLine_OUT].eMBRTUDeviceType = E_MBRTUMaster_DeviceType.eDrexelAWeiss_AereosilentStratosLU_Ventilation THEN
	//Aereosilent Stratos Ventilation Drexel and Weiss
	fbKL6xxxConfig.Mode := SERIALLINEMODE_KL6_22B_STANDARD;
	fbKL6xxxConfig.Baudrate := 19200;
	fbKL6xxxConfig.NoDatabits := 8;
	fbKL6xxxConfig.Parity := PARITY_NONE;
	fbKL6xxxConfig.Stopbits := 1;
	fbKL6xxxConfig.Handshake := HANDSHAKE_NONE;
	fbKL6xxxConfig.ContinousMode := FALSE;
	//Timout	
	timTimout.PT := T#10S;
	fbmodbusmaster.Timeout := T#3S;
ELSIF Lynus_Standards.GVL_Bussystems.stDataOfMBRTUMasterKL6xxx[diNrOfMBRTUMasterLine_OUT].eMBRTUDeviceType = E_MBRTUMaster_DeviceType.eABB_CM_UFD_M31M_NAProtection THEN
	//CM_UFD_M31M ABB NA Protection
	fbKL6xxxConfig.Mode := SERIALLINEMODE_KL6_22B_STANDARD;
	fbKL6xxxConfig.Baudrate := 38400;
	fbKL6xxxConfig.NoDatabits := 8;
	fbKL6xxxConfig.Parity := PARITY_NONE;
	fbKL6xxxConfig.Stopbits := 1;
	fbKL6xxxConfig.Handshake := RS485_HALFDUPLEX;
	fbKL6xxxConfig.ContinousMode := FALSE;
	//Timout	
	timTimout.PT := T#2S;
	fbmodbusmaster.Timeout := T#1S;
ELSIF Lynus_Standards.GVL_Bussystems.stDataOfMBRTUMasterKL6xxx[diNrOfMBRTUMasterLine_OUT].eMBRTUDeviceType = E_MBRTUMaster_DeviceType.eSchrack_ECS_CIONHOME_SEMIPUBLIC THEN
	//Schrack Electric Charging Station CionHome and Semipublic
	fbKL6xxxConfig.Mode := SERIALLINEMODE_KL6_22B_STANDARD;
	fbKL6xxxConfig.Baudrate := 57600;
	fbKL6xxxConfig.NoDatabits := 8;
	fbKL6xxxConfig.Parity := PARITY_NONE;
	fbKL6xxxConfig.Stopbits := 1;
	fbKL6xxxConfig.Handshake := RS485_HALFDUPLEX;
	fbKL6xxxConfig.ContinousMode := FALSE;
	//Timout	
	timTimout.PT := T#2S;
	fbmodbusmaster.Timeout := T#2S;
ELSIF Lynus_Standards.GVL_Bussystems.stDataOfMBRTUMasterKL6xxx[diNrOfMBRTUMasterLine_OUT].eMBRTUDeviceType = E_MBRTUMaster_DeviceType.ePV_DeltaSunspec THEN
	//Delte PV Inverter with Sunspec Protocol
	fbKL6xxxConfig.Mode := SERIALLINEMODE_KL6_22B_STANDARD;
	fbKL6xxxConfig.Baudrate := 19200;
	fbKL6xxxConfig.NoDatabits := 8;
	fbKL6xxxConfig.Parity := PARITY_NONE;
	fbKL6xxxConfig.Stopbits := 1;
	fbKL6xxxConfig.Handshake := RS485_HALFDUPLEX;
	fbKL6xxxConfig.ContinousMode := FALSE;
	//Timout	
	timTimout.PT := T#2S;
	fbmodbusmaster.Timeout := T#2S;
END_IF

FPConfigManual(CLK:= bConfigTerminal, Q=> );

fbKL6xxxConfig(
	Execute:= (FPConfigAuto.Q AND NOT bTerminalIsConfigured) OR (timInit.Q AND NOT bTerminalIsConfigured AND FPConfigManual.Q), 
	Mode:= ,
	Baudrate:= , 
	NoDatabits:= , 
	Parity:= , 
	Stopbits:= , 
	Handshake:= , 
	ContinousMode:= , 
	pComIn:= ADR(fbmodbusmaster.InData), 
	pComOut:= ADR(fbmodbusmaster.OutData), 
	SizeComIn:= SIZEOF(fbmodbusmaster.InData),
	Done=> , 
	Busy=> , 
	Error=> , 
	ErrorId=> );

IF fbKL6xxxConfig.Done THEN
	bTerminalIsConfigured := TRUE;
END_IF

(*------------------------------------------------------------------Read-Write----------------------------------------------------------------------------*)
	 
//Choose the right Modbus RTU Action for Read or Write Data
IF Lynus_Standards.GVL_Bussystems.stDataOfMBRTUMasterKL6xxx[diNrOfMBRTUMasterLine_OUT].eMBRTUReadWriteMode = E_MBRTUMaster_ReadWriteMode.eModbusRTUMaster_Diagnostics THEN 
	fbmodbusmaster.Diagnostics(); 
		fbmodbusmaster.cbLength := SIZEOF(Lynus_Standards.GVL_Bussystems.stDataOfMBRTUMasterKL6xxx[diNrOfMBRTUMasterLine_OUT].arrWriteOutData);
			fbmodbusmaster.pMemoryAddr := ADR(Lynus_Standards.GVL_Bussystems.stDataOfMBRTUMasterKL6xxx[diNrOfMBRTUMasterLine_OUT].arrWriteOutData);
END_IF
IF Lynus_Standards.GVL_Bussystems.stDataOfMBRTUMasterKL6xxx[diNrOfMBRTUMasterLine_OUT].eMBRTUReadWriteMode = E_MBRTUMaster_ReadWriteMode.eModbusRTUMaster_ReadCoils THEN 
	fbmodbusmaster.ReadCoils(); 
		fbmodbusmaster.cbLength := SIZEOF(arrRead);
			fbmodbusmaster.pMemoryAddr := ADR(arrRead);	
END_IF
IF Lynus_Standards.GVL_Bussystems.stDataOfMBRTUMasterKL6xxx[diNrOfMBRTUMasterLine_OUT].eMBRTUReadWriteMode = E_MBRTUMaster_ReadWriteMode.eModbusRTUMaster_ReadInputRegs THEN 
	fbmodbusmaster.ReadInputRegs(); 
		fbmodbusmaster.cbLength := SIZEOF(arrRead);
			fbmodbusmaster.pMemoryAddr := ADR(arrRead);
END_IF
IF Lynus_Standards.GVL_Bussystems.stDataOfMBRTUMasterKL6xxx[diNrOfMBRTUMasterLine_OUT].eMBRTUReadWriteMode = E_MBRTUMaster_ReadWriteMode.eModbusRTUMaster_ReadInputStatus THEN 
	fbmodbusmaster.ReadInputStatus(); 
		fbmodbusmaster.cbLength := SIZEOF(arrRead);
			fbmodbusmaster.pMemoryAddr := ADR(arrRead);
END_IF
IF Lynus_Standards.GVL_Bussystems.stDataOfMBRTUMasterKL6xxx[diNrOfMBRTUMasterLine_OUT].eMBRTUReadWriteMode = E_MBRTUMaster_ReadWriteMode.eModbusRTUMaster_ReadRegs THEN 
	fbmodbusmaster.ReadRegs();
		fbmodbusmaster.cbLength := SIZEOF(arrRead);
			fbmodbusmaster.pMemoryAddr := ADR(arrRead); 
END_IF
IF Lynus_Standards.GVL_Bussystems.stDataOfMBRTUMasterKL6xxx[diNrOfMBRTUMasterLine_OUT].eMBRTUReadWriteMode = E_MBRTUMaster_ReadWriteMode.eModbusRTUMaster_WriteMultipleCoils THEN 
	fbmodbusmaster.WriteMultipleCoils();
		fbmodbusmaster.cbLength := SIZEOF(Lynus_Standards.GVL_Bussystems.stDataOfMBRTUMasterKL6xxx[diNrOfMBRTUMasterLine_OUT].arrWriteOutData);
			fbmodbusmaster.pMemoryAddr := ADR(Lynus_Standards.GVL_Bussystems.stDataOfMBRTUMasterKL6xxx[diNrOfMBRTUMasterLine_OUT].arrWriteOutData); 
END_IF
IF Lynus_Standards.GVL_Bussystems.stDataOfMBRTUMasterKL6xxx[diNrOfMBRTUMasterLine_OUT].eMBRTUReadWriteMode = E_MBRTUMaster_ReadWriteMode.eModbusRTUMaster_WriteRegs THEN 
	fbmodbusmaster.WriteRegs(); 
		fbmodbusmaster.cbLength := SIZEOF(Lynus_Standards.GVL_Bussystems.stDataOfMBRTUMasterKL6xxx[diNrOfMBRTUMasterLine_OUT].arrWriteOutData);
			fbmodbusmaster.pMemoryAddr := ADR(Lynus_Standards.GVL_Bussystems.stDataOfMBRTUMasterKL6xxx[diNrOfMBRTUMasterLine_OUT].arrWriteOutData);
END_IF
IF Lynus_Standards.GVL_Bussystems.stDataOfMBRTUMasterKL6xxx[diNrOfMBRTUMasterLine_OUT].eMBRTUReadWriteMode = E_MBRTUMaster_ReadWriteMode.eModbusRTUMaster_WriteSingleCoil THEN 
	fbmodbusmaster.WriteSingleCoil(); 
		fbmodbusmaster.cbLength := SIZEOF(Lynus_Standards.GVL_Bussystems.stDataOfMBRTUMasterKL6xxx[diNrOfMBRTUMasterLine_OUT].arrWriteOutData);
			fbmodbusmaster.pMemoryAddr := ADR(Lynus_Standards.GVL_Bussystems.stDataOfMBRTUMasterKL6xxx[diNrOfMBRTUMasterLine_OUT].arrWriteOutData);
END_IF
IF Lynus_Standards.GVL_Bussystems.stDataOfMBRTUMasterKL6xxx[diNrOfMBRTUMasterLine_OUT].eMBRTUReadWriteMode = E_MBRTUMaster_ReadWriteMode.eModbusRTUMaster_WriteSingleRegister THEN 
	fbmodbusmaster.WriteSingleRegister(); 
		fbmodbusmaster.cbLength := SIZEOF(Lynus_Standards.GVL_Bussystems.stDataOfMBRTUMasterKL6xxx[diNrOfMBRTUMasterLine_OUT].arrWriteOutData);
			fbmodbusmaster.pMemoryAddr := ADR(Lynus_Standards.GVL_Bussystems.stDataOfMBRTUMasterKL6xxx[diNrOfMBRTUMasterLine_OUT].arrWriteOutData);
END_IF

//Order the range of MB Adress when we have a change on that on the slave Functions
IF MEMCMP(ADR(arrMBAdress),ADR(Lynus_Standards.GVL_Bussystems.stDataOfMBRTUMasterKL6xxx[diNrOfMBRTUMasterLine_OUT].arrAllModbusSlaveAdresses),SIZEOF(Lynus_Standards.GVL_Bussystems.stDataOfMBRTUMasterKL6xxx[diNrOfMBRTUMasterLine_OUT].arrAllModbusSlaveAdresses)) <> 0 AND iStateSetMBAdress = 0 THEN
	iStateSetMBAdress := 1;
		bStopReadWrite := TRUE;
			MEMCPY(ADR(arrMBAdress),ADR(Lynus_Standards.GVL_Bussystems.stDataOfMBRTUMasterKL6xxx[diNrOfMBRTUMasterLine_OUT].arrAllModbusSlaveAdresses),SIZEOF(Lynus_Standards.GVL_Bussystems.stDataOfMBRTUMasterKL6xxx[diNrOfMBRTUMasterLine_OUT].arrAllModbusSlaveAdresses));
END_IF

CASE iStateSetMBAdress OF
	
	0://Init
		bStopReadWrite := FALSE;

	1://Set the Actual Adress in use to 0 and Clear old MB Adresses in Array
		bTakeActualAdress := FALSE;
			byActualAdressInUse := 0;
				bySearchMBAdress := 0;
					byPosInArrayMBAdress := 0;	

		FOR byLPMBAdress := 1 TO 247 BY 1 DO
			Lynus_Standards.GVL_Bussystems.stDataOfMBRTUMasterKL6xxx[diNrOfMBRTUMasterLine_OUT].arrAllModbusSlaveAdresses[byLPMBAdress] := 0;
		END_FOR 
			
			iStateSetMBAdress := 2;	
		
	2://Order the new Adresses from lowest to highest
		bySearchMBAdress := bySearchMBAdress + 1;
			bySearchMBAdress := LIMIT(1,bySearchMBAdress,247);			
	
		FOR byLPMBAdress := 1 TO 247 BY 1 DO
			IF arrMBAdress[byLPMBAdress] = bySearchMBAdress THEN
				byPosInArrayMBAdress := byPosInArrayMBAdress + 1;
					byPosInArrayMBAdress := LIMIT(1,byPosInArrayMBAdress,247);
						Lynus_Standards.GVL_Bussystems.stDataOfMBRTUMasterKL6xxx[diNrOfMBRTUMasterLine_OUT].arrAllModbusSlaveAdresses[byPosInArrayMBAdress] := arrMBAdress[byLPMBAdress]; 	
			END_IF
		END_FOR  
		
		//Done
		IF bySearchMBAdress >= 247 THEN 
			iStateSetMBAdress := 0;
				MEMCPY(ADR(arrMBAdress),ADR(Lynus_Standards.GVL_Bussystems.stDataOfMBRTUMasterKL6xxx[diNrOfMBRTUMasterLine_OUT].arrAllModbusSlaveAdresses),SIZEOF(Lynus_Standards.GVL_Bussystems.stDataOfMBRTUMasterKL6xxx[diNrOfMBRTUMasterLine_OUT].arrAllModbusSlaveAdresses));
		END_IF 
	
END_CASE

//Check the Modbus Adresses from each Slave Device
FPProcessCompleted(CLK:= Lynus_Standards.GVL_Bussystems.stDataOfMBRTUMasterKL6xxx[diNrOfMBRTUMasterLine_OUT].bReadWriteIsDone, Q=> );
	FPError(CLK:= fbmodbusmaster.Error, Q=> );

bySmallestAdress := 247;	
	FOR byLPSmallestAdress := 1 TO 247 BY 1 DO
		IF Lynus_Standards.GVL_Bussystems.stDataOfMBRTUMasterKL6xxx[diNrOfMBRTUMasterLine_OUT].arrAllModbusSlaveAdresses[byLPSmallestAdress] < bySmallestAdress AND Lynus_Standards.GVL_Bussystems.stDataOfMBRTUMasterKL6xxx[diNrOfMBRTUMasterLine_OUT].arrAllModbusSlaveAdresses[byLPSmallestAdress] <> 0 THEN bySmallestAdress := Lynus_Standards.GVL_Bussystems.stDataOfMBRTUMasterKL6xxx[diNrOfMBRTUMasterLine_OUT].arrAllModbusSlaveAdresses[byLPSmallestAdress]; END_IF
	END_FOR
byBiggestAdress := 0;
	FOR byLPBiggestAdress := 1 TO 247 BY 1 DO
		IF Lynus_Standards.GVL_Bussystems.stDataOfMBRTUMasterKL6xxx[diNrOfMBRTUMasterLine_OUT].arrAllModbusSlaveAdresses[byLPBiggestAdress] > byBiggestAdress THEN byBiggestAdress := Lynus_Standards.GVL_Bussystems.stDataOfMBRTUMasterKL6xxx[diNrOfMBRTUMasterLine_OUT].arrAllModbusSlaveAdresses[byLPBiggestAdress]; END_IF  
	END_FOR
//Take the Next Adress after the Read/write is done
IF FPProcessCompleted.Q OR FPError.Q THEN
	bTakeActualAdress := TRUE;
		FOR byLPActualAdress := 1 TO 247 BY 1 DO
			IF Lynus_Standards.GVL_Bussystems.stDataOfMBRTUMasterKL6xxx[diNrOfMBRTUMasterLine_OUT].arrAllModbusSlaveAdresses[byLPActualAdress] > byActualAdressInUse THEN 
				byActualAdressInUse := Lynus_Standards.GVL_Bussystems.stDataOfMBRTUMasterKL6xxx[diNrOfMBRTUMasterLine_OUT].arrAllModbusSlaveAdresses[byLPActualAdress]; 
					EXIT;
			END_IF
		END_FOR		
END_IF

//Count the Number of RTU Slaves
byNumberOfTotalSlaves := 0;
	FOR byLPNumbersOfTotalSlaves := 1 TO 247 BY 1 DO
		IF Lynus_Standards.GVL_Bussystems.stDataOfMBRTUMasterKL6xxx[diNrOfMBRTUMasterLine_OUT].arrAllModbusSlaveAdresses[byLPNumbersOfTotalSlaves] <> 0 THEN byNumberOfTotalSlaves := byNumberOfTotalSlaves + 1; END_IF
	END_FOR

FNInitSmall(CLK:= bySmallestAdress = 247, Q=> );

IF byActualAdressInUse <> byActualAdressInUse_CP THEN bAdressHasChanged := TRUE; byActualAdressInUse_CP := byActualAdressInUse; ELSE bAdressHasChanged := FALSE; END_IF 

IF ((FPError.Q OR FPProcessCompleted.Q) AND NOT bAdressHasChanged) OR FNInitSmall.Q OR bySmallestAdress = byBiggestAdress THEN byActualAdressInUse := bySmallestAdress; END_IF

timTimout(IN:= Lynus_Standards.GVL_Bussystems.stDataOfMBRTUMasterKL6xxx[diNrOfMBRTUMasterLine_OUT].bReadWriteIsDone, PT:= , Q=> , ET=> );

IF FPProcessCompleted.Q OR timTimout.Q THEN Lynus_Standards.GVL_Bussystems.stDataOfMBRTUMasterKL6xxx[diNrOfMBRTUMasterLine_OUT].bReadWriteIsDone := FALSE; END_IF

IF NOT bTakeActualAdress THEN 
	fbmodbusmaster.UnitID := bySmallestAdress;
ELSE
	fbmodbusmaster.UnitID := byActualAdressInUse;
END_IF

fbmodbusmaster(
	UnitID:= , 
	Quantity:= Lynus_Standards.GVL_Bussystems.stDataOfMBRTUMasterKL6xxx[diNrOfMBRTUMasterLine_OUT].wNumberOfRegister, 
	MBAddr:= Lynus_Standards.GVL_Bussystems.stDataOfMBRTUMasterKL6xxx[diNrOfMBRTUMasterLine_OUT].wModbusRegister, 
	cbLength:= , 
	pMemoryAddr:= , 
	Execute:= Lynus_Standards.GVL_Bussystems.stDataOfMBRTUMasterKL6xxx[diNrOfMBRTUMasterLine_OUT].bSlaveStartReadOrWrite AND bTerminalIsConfigured AND NOT timDissableFunctions.Q AND NOT bStopReadWrite, 
	Timeout:= , 
	BUSY=> , 
	Error=> , 
	ErrorId=> , 
	cbRead=> );	
	
(*------------------------------------------------------------------Busy Flag----------------------------------------------------------------------------*)

IF NOT bTerminalIsConfigured THEN
	bBusy := fbKL6xxxConfig.Busy;
ELSE
	bBusy := fbmodbusmaster.BUSY;
END_IF

//When we have a change on the MB Adress List we set the Function always on Busy that al other Slave Functions Stops in the Init Step
IF bStopReadWrite THEN bBusy := TRUE; END_IF

FNBusy(CLK:= fbmodbusmaster.BUSY, Q=> );

(*------------------------------------------------------------------Error and Warning----------------------------------------------------------------------------*)

IF timDissableFunctions.Q THEN fbModbusRTUMessage.bWarning := TRUE; fbModbusRTUMessage.iWarningCode := 0; ELSE fbModbusRTUMessage.bWarning := FALSE; END_IF   
	IF (Lynus_Standards.GVL_Bussystems.diNumberOfMBRTUMasters > Constants_Bussystems.diMaxNumberOfMBRTUMasterKL6xxx) OR (NOT bTerminalIsConfigured AND fbKL6xxxConfig.Error) OR (bTerminalIsConfigured AND fbmodbusmaster.Error) OR bStopReadWrite THEN 
		fbModbusRTUMessage.bError := TRUE;
	ELSE
		fbModbusRTUMessage.bError := FALSE;
	END_IF

IF Lynus_Standards.GVL_Bussystems.diNumberOfMBRTUMasters > Constants_Bussystems.diMaxNumberOfMBRTUMasterKL6xxx THEN
	fbModbusRTUMessage.iErrorCode := 1;	
ELSIF NOT bTerminalIsConfigured THEN 
	IF fbKL6xxxConfig.Error THEN 
		fbModbusRTUMessage.iErrorCode := 2; 
	END_IF
//When we have a change on the MB Adress List we set the Function always on Error that al other Slave Functions go back to the Init Step
ELSIF bStopReadWrite THEN
	fbModbusRTUMessage.iErrorCode := 2; 
ELSE
	IF fbmodbusmaster.ErrorId = 1 THEN fbModbusRTUMessage.iErrorCode := 3; END_IF
	IF fbmodbusmaster.ErrorId = 2 THEN fbModbusRTUMessage.iErrorCode := 4; END_IF
	IF fbmodbusmaster.ErrorId = 3 THEN fbModbusRTUMessage.iErrorCode := 5; END_IF
	IF fbmodbusmaster.ErrorId = 4 THEN fbModbusRTUMessage.iErrorCode := 6; END_IF
	IF fbmodbusmaster.ErrorId = 5 THEN fbModbusRTUMessage.iErrorCode := 7; END_IF
	IF fbmodbusmaster.ErrorId = 6 THEN fbModbusRTUMessage.iErrorCode := 8; END_IF
	IF fbmodbusmaster.ErrorId = 7 THEN fbModbusRTUMessage.iErrorCode := 9; END_IF
	IF fbmodbusmaster.ErrorId = 8 THEN fbModbusRTUMessage.iErrorCode := 10; END_IF
	IF fbmodbusmaster.ErrorId = 16#A THEN fbModbusRTUMessage.iErrorCode := 11; END_IF
	IF fbmodbusmaster.ErrorId = 16#B THEN fbModbusRTUMessage.iErrorCode := 12; END_IF
	IF fbmodbusmaster.ErrorId = 16#20 THEN fbModbusRTUMessage.iErrorCode := 13; END_IF
	IF fbmodbusmaster.ErrorId = 16#21 THEN fbModbusRTUMessage.iErrorCode := 14; END_IF
	IF fbmodbusmaster.ErrorId = 16#22 THEN fbModbusRTUMessage.iErrorCode := 15; END_IF
	IF fbmodbusmaster.ErrorId = 16#23 THEN fbModbusRTUMessage.iErrorCode := 16; END_IF
	IF fbmodbusmaster.ErrorId = 16#24 THEN fbModbusRTUMessage.iErrorCode := 17; END_IF
	IF fbmodbusmaster.ErrorId = 16#25 THEN fbModbusRTUMessage.iErrorCode := 18; END_IF
	IF fbmodbusmaster.ErrorId = 102 THEN fbModbusRTUMessage.iErrorCode := 19; END_IF
	IF fbmodbusmaster.ErrorId = 103 THEN fbModbusRTUMessage.iErrorCode := 20; END_IF
	IF fbmodbusmaster.ErrorId = 107 THEN fbModbusRTUMessage.iErrorCode := 21; END_IF
	IF fbmodbusmaster.ErrorId = 110 THEN fbModbusRTUMessage.iErrorCode := 22; END_IF
	IF fbmodbusmaster.ErrorId = 120 THEN fbModbusRTUMessage.iErrorCode := 23; END_IF
	IF fbmodbusmaster.ErrorId = 150 THEN fbModbusRTUMessage.iErrorCode := 24; END_IF
	IF fbmodbusmaster.ErrorId = 232 THEN fbModbusRTUMessage.iErrorCode := 25; END_IF
	IF fbmodbusmaster.ErrorId = 233 THEN fbModbusRTUMessage.iErrorCode := 26; END_IF
END_IF

fbModbusRTUMessage(
	bTerminalConfigured:= bTerminalIsConfigured, 
	bError:= , 
	bWarning:= , 
	iWarningCode:= , 
	iErrorCode:= , 
	byErrorWarning=> byErrorWarning, 
	eMessageMBRTUMaster=> eMessageMBRTUMaster);

//Set this Flag after a Error and Reset after next Read or Write command without Error	
IF FPError.Q THEN bErrorIsActive := TRUE; END_IF
	IF FNBusy.Q AND NOT fbmodbusmaster.Error THEN bErrorIsActive := FALSE; END_IF	
	
FPErrorIsActive(CLK:= bErrorIsActive, Q=> );
	
(*-----------------------------------------------------------Handle data to Global structure for Modbus RTU Communication-----------------------------------------------------------------*)

CASE iStateGVLData OF
	
	0://Init Step
		byWaitInStep := 0;
			diCounterForGVL := 1;
	
	1://Wait for 4 Steps before clean al Data on GVL
		byWaitInStep := byWaitInStep + 1;
			IF byWaitInStep >= 4 AND fbNumberDevice.bNumberIsCalculatet THEN iStateGVLData := 2; END_IF
				//To much Devices, back to the Init step
				IF byWaitInStep >= 4 AND NOT fbNumberDevice.bNumberIsCalculatet THEN iStateGVLData := 0; END_IF	
			
	2://Clear all Data in GVL
	//Some Parts in the GVL Reset the Slave. Otherwise there will be problems when writing the new addresses to the array in the GVL.
	Lynus_Standards.GVL_Bussystems.stDataOfMBRTUMasterKL6xxx[diCounterForGVL].bMasterIsBusy := FALSE;	
		Lynus_Standards.GVL_Bussystems.stDataOfMBRTUMasterKL6xxx[diCounterForGVL].bTerminalIsConfigured := FALSE;	
			Lynus_Standards.GVL_Bussystems.stDataOfMBRTUMasterKL6xxx[diCounterForGVL].byNumberOfSlaves := 0;
				Lynus_Standards.GVL_Bussystems.stDataOfMBRTUMasterKL6xxx[diCounterForGVL].byErrorWarning := 0;
					Lynus_Standards.GVL_Bussystems.stDataOfMBRTUMasterKL6xxx[diCounterForGVL].byActualMBAdressInProgrss := 0;
						Lynus_Standards.GVL_Bussystems.stDataOfMBRTUMasterKL6xxx[diCounterForGVL].bNoNewMBusAdress := FALSE;	
														 		
		diCounterForGVL := diCounterForGVL + 1;
			diCounterForGVL := LIMIT(0,diCounterForGVL,Constants_Bussystems.diMaxNumberOfMBRTUMasterKL6xxx);
				//Back to the init step
				IF diCounterForGVL >= Constants_Bussystems.diMaxNumberOfMBRTUMasterKL6xxx THEN iStateGVLData := 0; END_IF

END_CASE 
	
IF diNrOfMBRTUMasterLine_OUT > 0 AND fbNumberDevice.bNumberIsCalculatet THEN  
	Lynus_Standards.GVL_Bussystems.stDataOfMBRTUMasterKL6xxx[diNrOfMBRTUMasterLine_OUT].bMasterIsBusy := bBusy;
		Lynus_Standards.GVL_Bussystems.stDataOfMBRTUMasterKL6xxx[diNrOfMBRTUMasterLine_OUT].byErrorWarning := byErrorWarning;
			Lynus_Standards.GVL_Bussystems.stDataOfMBRTUMasterKL6xxx[diNrOfMBRTUMasterLine_OUT].bTerminalIsConfigured := bTerminalIsConfigured;
				Lynus_Standards.GVL_Bussystems.stDataOfMBRTUMasterKL6xxx[diNrOfMBRTUMasterLine_OUT].byActualMBAdressInProgrss := fbmodbusmaster.UnitID;
					Lynus_Standards.GVL_Bussystems.stDataOfMBRTUMasterKL6xxx[diNrOfMBRTUMasterLine_OUT].byNumberOfSlaves := byNumberOfTotalSlaves;
						Lynus_Standards.GVL_Bussystems.stDataOfMBRTUMasterKL6xxx[diCounterForGVL].bNoNewMBusAdress := bStopReadWrite;
						IF FNBusy.Q THEN
							IF NOT fbmodbusmaster.Error THEN
								Lynus_Standards.GVL_Bussystems.stDataOfMBRTUMasterKL6xxx[diNrOfMBRTUMasterLine_OUT].arrReadOutData := arrRead;
							ELSE
								//Workarround about internal Beckhoff Lib Error 
								IF FPErrorIsActive.Q THEN 
									MEMCPY(ADR(fbmodbusmaster),ADR(fbmodbusmaster_Init),SIZEOF(fbmodbusmaster_Init));
								END_IF
							END_IF
						END_IF	
END_IF	
	
(*----------------------------------------------------------Save persistent data----------------------------------------------------------------*)

arrPD[1](lrValue:= BOOL_TO_LREAL(bTerminalIsConfigured), bEventBasedActive=> );
arrPD[2](lrValue:= INT_TO_LREAL(eDeviceType), bEventBasedActive=> );

END_FUNCTION_BLOCK

// ---- FBs/Schrack/FB_ECS_Schrack_EM_CionHome.TcPOU
FUNCTION_BLOCK FB_ECS_Schrack_EM_CionHome
VAR_INPUT PERSISTENT
	bEnable										: BOOL;																			//{#lynus.ag#()} //Enable the Fuctionblock and his logic
	bPowerDataInvers							: BOOL;																			//With True its possible to invert all received power data from the electric meter
	byElectricFuseLine							: BYTE; 																		//Electric Fuse Line on wich the ECS is connected => 1 2 3 (If 0 then this charging station is not connected to a Electric Fuse Line)
	byMBAdress									: BYTE;																			//The Modbus Adress from the Slave
	diNrOfMBRTUMasterLine_IN					: DINT;																			//Number of the RTU Master Function on what this function can send or write data
	diNrOfEMS_IN								: DINT;																			//Number of EMS what control this Device.
	diNrOfEM_IN_CS								: DINT;																			//Number of the electric meter for incoming power data. (Power Data for this Device)
	stSetupECS									: ST_Setup_ECS;																	//{#lynus.ag#()} //Setup charging station
END_VAR
VAR_OUTPUT
	stDataECS									: ST_ECS_Output;																//{#lynus.ag#()} //Electric charging station output data
	eSchrackErrors								: E_Schrack_ECS_Error;															//Error List of the Schrack charging station
	diNrOfECS_OUT								: DINT;																			//Active Number from the Electric charging Function for using on other functions
END_VAR
VAR
	{attribute 'hide'}
	fbCS										: FB_ElectricChargingStation;													//Function block for electric charging station
	{attribute 'hide'}
	fbNumberDevice								: FB_NumberOfDevice;															//Function block to calcualte the number of the Device
	fbDIExternalLock							: FB_XL1XXX_DI;																	//Digital Input from external loock signal
	{attribute 'hide'}
	fbCVChargingTime							: FB_CV_WORD_TO_DWORD;															//Convert the 2 word in a real type
	{attribute 'hide'}
	timDelay									: TON;																			//Timer for Delay between Requests
	{attribute 'hide'}
	timTimeout									: TON;																			//Timer for Timeout
	{attribute 'hide'}
	timDissableFunctions						: TON;																			//Timer to dissable the Function after Lynus_Standards.Constants_General.tTimeDissableLynusFunctions Days without connection to the Lynus Cloud
	{attribute 'hide'}
	timResetConnectionOnGVL						: TON;																			//Timer to try reset the connection Flag on the GVL. (When somebody delete the Connection Function and make only a onlinechange)
	{attribute 'hide'}
	timResetCS									: TOF;																			//Timer to send every 60 minutes a Reset command
	{attribute 'hide'}
	FPErrorMaster								: R_TRIG;																		//Internal positive Edge
	{attribute 'hide'}
	FPEnable									: R_TRIG;																		//Internal positive Edge
	{attribute 'hide'}
	FPChargingReleaseInvalid					: R_TRIG;																		//Internal positive Edge
	{attribute 'hide'}
	FPStateU									: R_TRIG;																		//Internal positive Edge
	{attribute 'hide'}
	FPResetCS									: R_TRIG;																		//Internal positive Edge
	{attribute 'hide'}
	FNError1CS									: F_TRIG;																		//Internal negative Edge
	{attribute 'hide'}
	FNError2CS									: F_TRIG;																		//Internal negative Edge
	{attribute 'hide'}
	FNError3CS									: F_TRIG;																		//Internal negative Edge
	{attribute 'hide'}
	arrPD										: ARRAY[1..18] OF FB_PersistentData_Number;										//Function to save persistent data
	{attribute 'hide'}
	arrErrorECS									: ARRAY[1..3] OF BOOL;															//Error from the ECS
	{attribute 'hide'}
	arrDefaultModbusAdress						: ARRAY[1..247] OF BYTE;														//Default Modbuss Adress Array to fill in in the GVL Array after a Online change
	{attribute 'hide'}
	arrDefaultReadWrite							: ARRAY[1..Constants_Bussystems.wQuantityOfRegistersMBRTUMaster] OF WORD;		//Default Read/Write Array to fill in in the GVL Array after a Online change
	{attribute 'hide'}
	arrCounterForGVL							: ARRAY[1..2] OF DINT;															//Counter to clean old data on GVL
	{attribute 'hide'}
	bChargeCableIsConnected						: BOOL;																			//Shows if the Charge cabel i sconnected to the ECS and the Car
	{attribute 'hide'}
	bAdressIsSet								: BOOL;																			//Its true when the new Modbus Adress from the Slave is set in the Array on the GVL for the Master	
	{attribute 'hide'}
	bChargingReleaseInavlid						: BOOL;																			//State of the charging release invalid	
	{attribute 'hide'}
	bResetCS									: BOOL;																			//Reset the charging station after a internal Charging station error or Charging Station Stae 16#55
	{attribute 'hide'}
	byWaitInStep								: BYTE;																			//Wait in Step before start to clean data on PLC
	{attribute 'hide'}
	byNumberOfSameMBAdress						: BYTE;																			//Number of Same Modbus adress on 1 Modbus Master
	{attribute 'hide'}
	byMBAdress_Old								: BYTE;																			//Old Modbus Adress to compare with the new Modbus Adress to start the state machine to set in the Array on the GVL
	{attribute 'hide'}
	byMBAdress_CP								: BYTE;																			//Variable to compare the Modbus Adress in the State Machine. When the Adress change when the state machine is active then the state machine starts from new with the new adress 
	{attribute 'hide'}
	byLPSlaveAdress								: BYTE;																			//Loop for the state machine to set the adress from the Slave in the array on the GVL
	{attribute 'hide'}
	iStateGVLData								: INT;																			//State machine to handle the data on the GVL
	{attribute 'hide'}
	iStateModbusRead							: INT;																			//State machine for read out Data over Modbus RTU
	{attribute 'hide'}
	iStateModbusWrite							: INT;																			//State machine for write Data over Modbus RTU
	{attribute 'hide'}
	iStateModbusError							: INT;																			//State machine for error out Data over Modbus RTU	
	{attribute 'hide'}
	iStateModbus_CP								: INT;																			//Variable to compare the state machine variable to set or reset the timeout timer
	{attribute 'hide'}
	wCPStateECS									: WORD;																			//CP State from th CS
	{attribute 'hide'}
	wLPCleanBuffer								: WORD;																			//Loop to clear the send and write Buffer on the GVL
	{attribute 'hide'}
	diNrOfMBRTUMasterLine_IN_Old				: DINT;																			//Old Modbus RTU Line to compare with the new Modbus RTU Line to start the state machine to set in the Array on the GVL
	{attribute 'hide'}
	diNrOfMBRTUMasterLine_IN_CP					: DINT;																			//Variable to compare the Modbus RTU Line in the State Machine. When the Modbus RTU Line change when the state machine is active then the state machine starts from new with the new Modbus RTU Line
	{attribute 'hide'}
	diNumberOfActiveBatterys					: DINT;																			//Number of active batterys
	{attribute 'hide'}
	diNumberOfBatteryInverterInEPO				: DINT;																			//Number of battery inverters that work in Emergency Power operation 
	{attribute 'hide'}
	diLPForGVL									: DINT;																			//Loop to clean old data on GVL
	{attribute 'hide'}
	dwSumSOC									: DWORD;																		//Sum of the SOC from all batterys
	{attribute 'hide'}	
	liLPBatteryData								: LINT;																			//Loop to check some data from batterys
	{attribute 'hide'}
	liLPInEPO									: LINT;																			//Loop to check if 1 or more battery inverters build a island grid
END_VAR
VAR PERSISTENT
	{attribute 'conditionalshow'}
	byMBAdress_ForChange						: BYTE;																			//When we have 2 same Adresses on 1 Modbus RTU Line the byMBAdress_Int is set to 0. After a other change on the Input Adress Field so we can start to set the Adress in the Array in the GVL
	byMBAdress_Int								: BYTE;																			//Internal Adress what is using for the Read and Write functions
	diNrOfEMS_IN_CP								: DINT;																			//Number of EMS what control this Device to compare with the original
END_VAR

//Creator : Kai Ebensperger
//Company : Lynus AG
//Date : 12.07.2021
//Version : 1.0.0.0

//With this Funcition its possible to communicate with a Schrack Electric charging station from the Cion Home and Semipublic Series over Modbus RTU.
//Runs with this ECS : EMCION11C-
//EMCION22C-
//EMCION22P-
//EMCION11CR
//EMCION22CR
//EMCION22PR
//Its possible to controll the charging station over the charg current
//This function set the minimal charge current from the charging station to 6 Ampere 
//When the Function send 0 Ampere or is switched of, then the charging station is blocked and its not possible to charge
//Versions that are supported : Date : 13.04.2021

//NOTE for diNr.....Designation => 
//_IN = Here Data come in from other Functions or go out to other functions about the GVL
//_OUT = Here Data go out to other functions about the GVL

(*--------------------------------------------------------------------------------------------Limits-------------------------------------------------------------------------------------*)

byMBAdress := LIMIT(0,byMBAdress,247);
	diNrOfMBRTUMasterLine_IN := LIMIT(0,diNrOfMBRTUMasterLine_IN,Constants_Bussystems.diMaxNumberOfMBRTUMasterKL6xxx);	
		diNrOfEMS_IN := LIMIT(0,diNrOfEMS_IN,Constants_Energy.diMaxNumberOfEMS);
			diNrOfEM_IN_CS := LIMIT(0,diNrOfEM_IN_CS,Constants_Energy.diMaxNumberOfElectricMeters);
				byElectricFuseLine := LIMIT(0,byElectricFuseLine,30);

(*------------------------------------------------------------------Power Data----------------------------------------------------------------------------*)

